LIN {X 0,Y 247.434,Z 446.734,A -85,B 0,C 180,E1 -19045.448,E2 -19045.448} C_VEL
LIN {X 0,Y 248.278,Z 445.373,A -85,B 0,C 180,E1 -19048.116,E2 -19048.116} C_VEL
LIN {X 0,Y 249.454,Z 442.811,A -85,B 0,C 180,E1 -19050.842,E2 -19050.842} C_VEL
LIN {X 0,Y 251.057,Z 438.873,A -85,B 0,C 180,E1 -19053.598,E2 -19053.598} C_VEL
LIN {X 0,Y 253.141,Z 433.443,A -85,B 0,C 180,E1 -19056.36,E2 -19056.36} C_VEL
LIN {X 0,Y 255.295,Z 427.674,A -85,B 0,C 180,E1 -19058.608,E2 -19058.608} C_VEL
LIN {X 0,Y 257.786,Z 420.296,A -85,B 0,C 180,E1 -19060.904,E2 -19060.904} C_VEL
LIN {X 0,Y 260.58,Z 411.115,A -85,B 0,C 180,E1 -19063.147,E2 -19063.147} C_VEL
LIN {X 0,Y 263.573,Z 400.733,A -85,B 0,C 180,E1 -19065.13,E2 -19065.13} C_VEL
LIN {X 0,Y 266.276,Z 389.982,A -85,B 0,C 180,E1 -19066.742,E2 -19066.742} C_VEL
LIN {X 0,Y 268.643,Z 378.487,A -85,B 0,C 180,E1 -19068.111,E2 -19068.111} C_VEL
LIN {X 0,Y 270.76,Z 365.913,A -85,B 0,C 180,E1 -19069.248,E2 -19069.248} C_VEL
LIN {X 0,Y 272.299,Z 353.044,A -85,B 0,C 180,E1 -19070.095,E2 -19070.095} C_VEL
LIN {X 0,Y 273.399,Z 340.201,A -85,B 0,C 180,E1 -19070.646,E2 -19070.646} C_VEL
LIN {X 0,Y 276.818,Z 284.839,A -85,B 0,C 180,E1 -19072.41,E2 -19072.41} C_VEL
LIN {X 0,Y 272.206,Z 274.812,A -85,B 0,C 180,E1 -19073.807,E2 -19073.807} C_VEL
LIN {X 0,Y 266.984,Z 265.08,A -85,B 0,C 180,E1 -19075.436,E2 -19075.436} C_VEL
LIN {X 0,Y 262.474,Z 257.861,A -85,B 0,C 180,E1 -19076.931,E2 -19076.931} C_VEL
LIN {X 0,Y 255.943,Z 247.889,A -85,B 0,C 180,E1 -19079.312,E2 -19079.312} C_VEL
LIN {X 0,Y 252.331,Z 243.094,A -85,B 0,C 180,E1 -19080.75,E2 -19080.75} C_VEL
LIN {X 0,Y 250.81,Z 241.467,A -85,B 0,C 180,E1 -19081.366,E2 -19081.366} C_VEL
LIN {X 0,Y 249.325,Z 240.348,A -85,B 0,C 180,E1 -19081.963,E2 -19081.963} C_VEL
LIN {X 0,Y 244.214,Z 240.449,A -85,B 0,C 180,E1 -19084.001,E2 -19084.001} C_VEL
LIN {X 0,Y 242.5,Z 239.911,A -85,B 0,C 180,E1 -19085.228,E2 -19085.228} C_VEL
LIN {X 0,Y 242.285,Z 239.3,A -85,B 0,C 180,E1 -19085.875,E2 -19085.875} C_VEL
LIN {X 0,Y 242.288,Z 239.303,A -85,B 0,C 180,E1 -19089.556,E2 -19089.556} C_VEL
LIN {X 0,Y 242.106,Z 239.323,A -85,B 0,C 180,E1 -19093.429,E2 -19093.429} C_VEL
LIN {X 0,Y 242.079,Z 239.323,A -85,B 0,C 180,E1 -19096.878,E2 -19096.878} C_VEL
LIN {X 0,Y 241.965,Z 239.346,A -85,B 0,C 180,E1 -19102.185,E2 -19102.185} C_VEL
LIN {X 0,Y 242.03,Z 239.332,A -85,B 0,C 180,E1 -19105.832,E2 -19105.832} C_VEL
LIN {X 0,Y 241.955,Z 239.338,A -85,B 0,C 180,E1 -19109.591,E2 -19109.591} C_VEL
LIN {X 0,Y 241.95,Z 239.343,A -85,B 0,C 180,E1 -19113.498,E2 -19113.498} C_VEL
LIN {X 0,Y 241.978,Z 239.412,A -85,B 0,C 180,E1 -19118.102,E2 -19118.102} C_VEL
LIN {X 0,Y 243.913,Z 244.836,A -85,B 0,C 180,E1 -19122.62,E2 -19122.62} C_VEL
LIN {X 0,Y 246.041,Z 251.254,A -85,B 0,C 180,E1 -19126.866,E2 -19126.866} C_VEL
LIN {X 0,Y 249.47,Z 256.649,A -85,B 0,C 180,E1 -19128.448,E2 -19128.448} C_VEL
LIN {X 0,Y 250.911,Z 258.872,A -85,B 0,C 180,E1 -19129.069,E2 -19129.069} C_VEL
LIN {X 0,Y 254.41,Z 264.527,A -85,B 0,C 180,E1 -19130.496,E2 -19130.496} C_VEL
LIN {X 0,Y 257.98,Z 270.888,A -85,B 0,C 180,E1 -19131.875,E2 -19131.875} C_VEL
LIN {X 0,Y 262.221,Z 279.028,A -85,B 0,C 180,E1 -19133.4,E2 -19133.4} C_VEL
LIN {X 0,Y 267,Z 289.735,A -85,B 0,C 180,E1 -19135.057,E2 -19135.057} C_VEL
LIN {X 0,Y 267.899,Z 292.556,A -85,B 0,C 180,E1 -19135.388,E2 -19135.388} C_VEL
LIN {X 0,Y 269.758,Z 308.366,A -85,B 0,C 180,E1 -19136.523,E2 -19136.523} C_VEL
LIN {X 0,Y 270.142,Z 313.745,A -85,B 0,C 180,E1 -19136.851,E2 -19136.851} C_VEL
LIN {X 0,Y 266.746,Z 363.722,A -85,B 0,C 180,E1 -19138.482,E2 -19138.482} C_VEL
LIN {X 0,Y 265.058,Z 377.664,A -85,B 0,C 180,E1 -19139.202,E2 -19139.202} C_VEL
LIN {X 0,Y 262.799,Z 390.364,A -85,B 0,C 180,E1 -19140.13,E2 -19140.13} C_VEL
LIN {X 0,Y 260.117,Z 402.51,A -85,B 0,C 180,E1 -19141.345,E2 -19141.345} C_VEL
LIN {X 0,Y 257.264,Z 413.548,A -85,B 0,C 180,E1 -19142.772,E2 -19142.772} C_VEL
LIN {X 0,Y 254.38,Z 423.635,A -85,B 0,C 180,E1 -19144.428,E2 -19144.428} C_VEL
LIN {X 0,Y 251.149,Z 433.64,A -85,B 0,C 180,E1 -19146.502,E2 -19146.502} C_VEL
LIN {X 0,Y 248.189,Z 442.707,A -85,B 0,C 180,E1 -19148.881,E2 -19148.881} C_VEL
LIN {X 0,Y 245.728,Z 449.849,A -85,B 0,C 180,E1 -19151.256,E2 -19151.256} C_VEL
LIN {X 0,Y 244.09,Z 454.725,A -85,B 0,C 180,E1 -19153.268,E2 -19153.268} C_VEL
LIN {X 0,Y 242.262,Z 459.556,A -85,B 0,C 180,E1 -19155.726,E2 -19155.726} C_VEL
LIN {X 0,Y 241.102,Z 463.286,A -85,B 0,C 180,E1 -19158.228,E2 -19158.228} C_VEL
LIN {X 0,Y 240.531,Z 465.241,A -85,B 0,C 180,E1 -19159.904,E2 -19159.904} C_VEL
LIN {X 0,Y 239.9,Z 467.837,A -85,B 0,C 180,E1 -19163.271,E2 -19163.271} C_VEL
LIN {X 0,Y 239.811,Z 468.612,A -85,B 0,C 180,E1 -19165.156,E2 -19165.156} C_VEL
LIN {X 0,Y 239.87,Z 468.846,A -85,B 0,C 180,E1 -19166.641,E2 -19166.641} C_VEL
LIN {X 0,Y 239.974,Z 468.704,A -85,B 0,C 180,E1 -19168.322,E2 -19168.322} C_VEL
LIN {X 0,Y 240.024,Z 468.154,A -85,B 0,C 180,E1 -19170,E2 -19170} C_VEL
LIN {X 0,Y 240.005,Z 467.189,A -85,B 0,C 180,E1 -19171.678,E2 -19171.678} C_VEL
LIN {X 0,Y 239.998,Z 465.777,A -85,B 0,C 180,E1 -19173.357,E2 -19173.357} C_VEL
LIN {X 0,Y 240.032,Z 463.373,A -85,B 0,C 180,E1 -19175.432,E2 -19175.432} C_VEL
LIN {X 0,Y 240.199,Z 458.645,A -85,B 0,C 180,E1 -19178.411,E2 -19178.411} C_VEL
LIN {X 0,Y 240.795,Z 452.239,A -85,B 0,C 180,E1 -19181.361,E2 -19181.361} C_VEL
LIN {X 0,Y 241.75,Z 445.225,A -85,B 0,C 180,E1 -19183.875,E2 -19183.875} C_VEL
LIN {X 0,Y 242.768,Z 438.024,A -85,B 0,C 180,E1 -19185.961,E2 -19185.961} C_VEL
LIN {X 0,Y 244.201,Z 428.768,A -85,B 0,C 180,E1 -19188.136,E2 -19188.136} C_VEL
LIN {X 0,Y 245.718,Z 418.531,A -85,B 0,C 180,E1 -19190.071,E2 -19190.071} C_VEL
LIN {X 0,Y 247.301,Z 407.905,A -85,B 0,C 180,E1 -19191.679,E2 -19191.679} C_VEL
LIN {X 0,Y 248.892,Z 396.173,A -85,B 0,C 180,E1 -19193.063,E2 -19193.063} C_VEL
LIN {X 0,Y 250.367,Z 382.933,A -85,B 0,C 180,E1 -19194.235,E2 -19194.235} C_VEL
LIN {X 0,Y 251.516,Z 369.594,A -85,B 0,C 180,E1 -19195.053,E2 -19195.053} C_VEL
LIN {X 0,Y 252.294,Z 352.667,A -85,B 0,C 180,E1 -19195.688,E2 -19195.688} C_VEL
LIN {X 0,Y 253.806,Z 307.843,A -85,B 0,C 180,E1 -19197.169,E2 -19197.169} C_VEL
LIN {X 0,Y 248.709,Z 266.187,A -85,B 0,C 180,E1 -19199.124,E2 -19199.124} C_VEL
LIN {X 0,Y 245.747,Z 257.13,A -85,B 0,C 180,E1 -19199.767,E2 -19199.767} C_VEL
LIN {X 0,Y 243.216,Z 244.807,A -85,B 0,C 180,E1 -19204.291,E2 -19204.291} C_VEL
LIN {X 0,Y 242.051,Z 239.335,A -85,B 0,C 180,E1 -19206.417,E2 -19206.417} C_VEL
LIN {X 0,Y 241.91,Z 239.35,A -85,B 0,C 180,E1 -19210.943,E2 -19210.943} C_VEL
LIN {X 0,Y 241.905,Z 239.355,A -85,B 0,C 180,E1 -19214.201,E2 -19214.201} C_VEL
LIN {X 0,Y 241.915,Z 239.352,A -85,B 0,C 180,E1 -19218.072,E2 -19218.072} C_VEL
LIN {X 0,Y 241.971,Z 239.342,A -85,B 0,C 180,E1 -19222.414,E2 -19222.414} C_VEL
LIN {X 0,Y 241.949,Z 239.343,A -85,B 0,C 180,E1 -19226.502,E2 -19226.502} C_VEL
LIN {X 0,Y 241.964,Z 239.343,A -85,B 0,C 180,E1 -19230.607,E2 -19230.607} C_VEL
LIN {X 0,Y 242.029,Z 239.331,A -85,B 0,C 180,E1 -19234.178,E2 -19234.178} C_VEL
LIN {X 0,Y 241.968,Z 239.343,A -85,B 0,C 180,E1 -19238.332,E2 -19238.332} C_VEL
LIN {X 0,Y 242.089,Z 239.32,A -85,B 0,C 180,E1 -19243.316,E2 -19243.316} C_VEL
LIN {X 0,Y 242.138,Z 239.32,A -85,B 0,C 180,E1 -19248.277,E2 -19248.277} C_VEL
LIN {X 0,Y 242.363,Z 239.294,A -85,B 0,C 180,E1 -19251.663,E2 -19251.663} C_VEL
LIN {X 0,Y 242.386,Z 239.29,A -85,B 0,C 180,E1 -19253.339,E2 -19253.339} C_VEL
LIN {X 0,Y 242.599,Z 239.251,A -85,B 0,C 180,E1 -19258.339,E2 -19258.339} C_VEL
LIN {X 0,Y 242.601,Z 239.255,A -85,B 0,C 180,E1 -19261.659,E2 -19261.659} C_VEL
LIN {X 0,Y 242.379,Z 239.292,A -85,B 0,C 180,E1 -19266.797,E2 -19266.797} C_VEL
LIN {X 0,Y 242.234,Z 239.309,A -85,B 0,C 180,E1 -19270.024,E2 -19270.024} C_VEL
LIN {X 0,Y 242.112,Z 239.314,A -85,B 0,C 180,E1 -19275.144,E2 -19275.144} C_VEL
LIN {X 0,Y 242.057,Z 239.312,A -85,B 0,C 180,E1 -19278.625,E2 -19278.625} C_VEL
LIN {X 0,Y 242.049,Z 239.322,A -85,B 0,C 180,E1 -19282.176,E2 -19282.176} C_VEL
LIN {X 0,Y 242.044,Z 239.33,A -85,B 0,C 180,E1 -19285.84,E2 -19285.84} C_VEL
LIN {X 0,Y 242.007,Z 239.337,A -85,B 0,C 180,E1 -19289.583,E2 -19289.583} C_VEL
LIN {X 0,Y 241.96,Z 239.34,A -85,B 0,C 180,E1 -19293.495,E2 -19293.495} C_VEL
LIN {X 0,Y 241.98,Z 239.329,A -85,B 0,C 180,E1 -19297.583,E2 -19297.583} C_VEL
LIN {X 0,Y 241.964,Z 239.331,A -85,B 0,C 180,E1 -19301.916,E2 -19301.916} C_VEL
LIN {X 0,Y 241.921,Z 239.347,A -85,B 0,C 180,E1 -19305.802,E2 -19305.802} C_VEL
LIN {X 0,Y 241.943,Z 239.347,A -85,B 0,C 180,E1 -19310.284,E2 -19310.284} C_VEL
LIN {X 0,Y 241.976,Z 239.335,A -85,B 0,C 180,E1 -19314.492,E2 -19314.492} C_VEL
LIN {X 0,Y 241.965,Z 239.333,A -85,B 0,C 180,E1 -19318.483,E2 -19318.483} C_VEL
LIN {X 0,Y 242.003,Z 239.338,A -85,B 0,C 180,E1 -19322.316,E2 -19322.316} C_VEL
LIN {X 0,Y 242.051,Z 239.334,A -85,B 0,C 180,E1 -19326.018,E2 -19326.018} C_VEL
LIN {X 0,Y 242.032,Z 239.331,A -85,B 0,C 180,E1 -19329.61,E2 -19329.61} C_VEL
LIN {X 0,Y 242.159,Z 239.316,A -85,B 0,C 180,E1 -19333.28,E2 -19333.28} C_VEL
LIN {X 0,Y 242.184,Z 239.314,A -85,B 0,C 180,E1 -19338.281,E2 -19338.281} C_VEL
LIN {X 0,Y 242.424,Z 239.287,A -85,B 0,C 180,E1 -19341.667,E2 -19341.667} C_VEL
LIN {X 0,Y 242.257,Z 239.31,A -85,B 0,C 180,E1 -19345.008,E2 -19345.008} C_VEL
LIN {X 0,Y 242.635,Z 239.258,A -85,B 0,C 180,E1 -19348.341,E2 -19348.341} C_VEL
LIN {X 0,Y 242.635,Z 239.259,A -85,B 0,C 180,E1 -19351.66,E2 -19351.66} C_VEL
LIN {X 0,Y 242.423,Z 239.287,A -85,B 0,C 180,E1 -19356.659,E2 -19356.659} C_VEL
LIN {X 0,Y 242.265,Z 239.307,A -85,B 0,C 180,E1 -19360.023,E2 -19360.023} C_VEL
LIN {X 0,Y 242.163,Z 239.322,A -85,B 0,C 180,E1 -19365.139,E2 -19365.139} C_VEL
LIN {X 0,Y 242.067,Z 239.332,A -85,B 0,C 180,E1 -19369.503,E2 -19369.503} C_VEL
LIN {X 0,Y 242.098,Z 239.466,A -85,B 0,C 180,E1 -19370.163,E2 -19370.163} C_VEL
LIN {X 0,Y 247.724,Z 253.276,A -85,B 0,C 180,E1 -19371.215,E2 -19371.215} C_VEL
LIN {X 0,Y 253.573,Z 269.164,A -85,B 0,C 180,E1 -19372.309,E2 -19372.309} C_VEL
LIN {X 0,Y 254.862,Z 273.057,A -85,B 0,C 180,E1 -19372.559,E2 -19372.559} C_VEL
LIN {X 0,Y 252.021,Z 343.618,A -85,B 0,C 180,E1 -19374.889,E2 -19374.889} C_VEL
LIN {X 0,Y 251.08,Z 357.249,A -85,B 0,C 180,E1 -19375.654,E2 -19375.654} C_VEL
LIN {X 0,Y 250.037,Z 370.169,A -85,B 0,C 180,E1 -19376.723,E2 -19376.723} C_VEL
LIN {X 0,Y 248.619,Z 382.874,A -85,B 0,C 180,E1 -19378.143,E2 -19378.143} C_VEL
LIN {X 0,Y 247.293,Z 393.032,A -85,B 0,C 180,E1 -19379.587,E2 -19379.587} C_VEL
LIN {X 0,Y 245.776,Z 403.642,A -85,B 0,C 180,E1 -19381.462,E2 -19381.462} C_VEL
LIN {X 0,Y 244.339,Z 412.802,A -85,B 0,C 180,E1 -19383.475,E2 -19383.475} C_VEL
LIN {X 0,Y 242.893,Z 421.687,A -85,B 0,C 180,E1 -19385.889,E2 -19385.889} C_VEL
LIN {X 0,Y 241.795,Z 428.792,A -85,B 0,C 180,E1 -19388.301,E2 -19388.301} C_VEL
LIN {X 0,Y 240.966,Z 434.411,A -85,B 0,C 180,E1 -19390.685,E2 -19390.685} C_VEL
LIN {X 0,Y 240.445,Z 438.85,A -85,B 0,C 180,E1 -19393.053,E2 -19393.053} C_VEL
LIN {X 0,Y 239.996,Z 442.182,A -85,B 0,C 180,E1 -19395.348,E2 -19395.348} C_VEL
LIN {X 0,Y 239.735,Z 444.602,A -85,B 0,C 180,E1 -19397.604,E2 -19397.604} C_VEL
LIN {X 0,Y 239.645,Z 446.243,A -85,B 0,C 180,E1 -19399.821,E2 -19399.821} C_VEL
LIN {X 0,Y 239.806,Z 447.23,A -85,B 0,C 180,E1 -19402.298,E2 -19402.298} C_VEL
LIN {X 0,Y 240.228,Z 447.289,A -85,B 0,C 180,E1 -19404.991,E2 -19404.991} C_VEL
LIN {X 0,Y 241.028,Z 446.267,A -85,B 0,C 180,E1 -19407.726,E2 -19407.726} C_VEL
LIN {X 0,Y 242.178,Z 444.088,A -85,B 0,C 180,E1 -19410.517,E2 -19410.517} C_VEL
LIN {X 0,Y 243.783,Z 440.637,A -85,B 0,C 180,E1 -19413.329,E2 -19413.329} C_VEL
LIN {X 0,Y 246.062,Z 435.194,A -85,B 0,C 180,E1 -19416.431,E2 -19416.431} C_VEL
LIN {X 0,Y 248.473,Z 429.163,A -85,B 0,C 180,E1 -19418.955,E2 -19418.955} C_VEL
LIN {X 0,Y 251.308,Z 421.317,A -85,B 0,C 180,E1 -19421.515,E2 -19421.515} C_VEL
LIN {X 0,Y 254.172,Z 412.662,A -85,B 0,C 180,E1 -19423.743,E2 -19423.743} C_VEL
LIN {X 0,Y 257.286,Z 402.561,A -85,B 0,C 180,E1 -19425.769,E2 -19425.769} C_VEL
LIN {X 0,Y 259.926,Z 392.988,A -85,B 0,C 180,E1 -19427.295,E2 -19427.295} C_VEL
LIN {X 0,Y 262.588,Z 381.11,A -85,B 0,C 180,E1 -19428.812,E2 -19428.812} C_VEL
LIN {X 0,Y 264.792,Z 369.498,A -85,B 0,C 180,E1 -19429.931,E2 -19429.931} C_VEL
LIN {X 0,Y 266.554,Z 356.371,A -85,B 0,C 180,E1 -19430.898,E2 -19430.898} C_VEL
LIN {X 0,Y 267.891,Z 342.608,A -85,B 0,C 180,E1 -19431.545,E2 -19431.545} C_VEL
LIN {X 0,Y 271.618,Z 287.449,A -85,B 0,C 180,E1 -19433.342,E2 -19433.342} C_VEL
LIN {X 0,Y 266.636,Z 276.755,A -85,B 0,C 180,E1 -19434.933,E2 -19434.933} C_VEL
LIN {X 0,Y 261.493,Z 267.258,A -85,B 0,C 180,E1 -19436.682,E2 -19436.682} C_VEL
LIN {X 0,Y 253.706,Z 254.952,A -85,B 0,C 180,E1 -19439.567,E2 -19439.567} C_VEL
LIN {X 0,Y 249.474,Z 249.158,A -85,B 0,C 180,E1 -19441.312,E2 -19441.312} C_VEL
LIN {X 0,Y 247.381,Z 246.516,A -85,B 0,C 180,E1 -19442.24,E2 -19442.24} C_VEL
LIN {X 0,Y 245.331,Z 244.219,A -85,B 0,C 180,E1 -19443.182,E2 -19443.182} C_VEL
LIN {X 0,Y 243.211,Z 242.091,A -85,B 0,C 180,E1 -19444.195,E2 -19444.195} C_VEL
LIN {X 0,Y 242.531,Z 240.662,A -85,B 0,C 180,E1 -19444.675,E2 -19444.675} C_VEL
LIN {X 0,Y 242.285,Z 239.3,A -85,B 0,C 180,E1 -19445.875,E2 -19445.875} C_VEL
LIN {X 0,Y 241.688,Z 239.381,A -85,B 0,C 180,E1 -19447.263,E2 -19447.263} C_VEL
LIN {X 0,Y 240.082,Z 239.578,A -85,B 0,C 180,E1 -19448.623,E2 -19448.623} C_VEL
LIN {X 0,Y 236.204,Z 240.055,A -85,B 0,C 180,E1 -19451.362,E2 -19451.362} C_VEL
LIN {X 0,Y 235.113,Z 240.199,A -85,B 0,C 180,E1 -19452.795,E2 -19452.795} C_VEL
LIN {X 0,Y 235.03,Z 240.199,A -85,B 0,C 180,E1 -19453.282,E2 -19453.282} C_VEL
LIN {X 0,Y 234.987,Z 240.206,A -85,B 0,C 180,E1 -19457.403,E2 -19457.403} C_VEL
LIN {X 0,Y 234.931,Z 240.223,A -85,B 0,C 180,E1 -19461.987,E2 -19461.987} C_VEL
LIN {X 0,Y 234.962,Z 240.21,A -85,B 0,C 180,E1 -19466.202,E2 -19466.202} C_VEL
LIN {X 0,Y 234.874,Z 240.223,A -85,B 0,C 180,E1 -19470.577,E2 -19470.577} C_VEL
LIN {X 0,Y 234.902,Z 240.364,A -85,B 0,C 180,E1 -19474.43,E2 -19474.43} C_VEL
LIN {X 0,Y 236.327,Z 244.216,A -85,B 0,C 180,E1 -19478.647,E2 -19478.647} C_VEL
LIN {X 0,Y 238.304,Z 249.77,A -85,B 0,C 180,E1 -19483.29,E2 -19483.29} C_VEL
LIN {X 0,Y 238.701,Z 250.699,A -85,B 0,C 180,E1 -19483.782,E2 -19483.782} C_VEL
LIN {X 0,Y 242.195,Z 255.987,A -85,B 0,C 180,E1 -19485.722,E2 -19485.722} C_VEL
LIN {X 0,Y 243.536,Z 257.884,A -85,B 0,C 180,E1 -19486.391,E2 -19486.391} C_VEL
LIN {X 0,Y 247.667,Z 264.331,A -85,B 0,C 180,E1 -19488.345,E2 -19488.345} C_VEL
LIN {X 0,Y 250.972,Z 269.919,A -85,B 0,C 180,E1 -19489.778,E2 -19489.778} C_VEL
LIN {X 0,Y 254.538,Z 276.479,A -85,B 0,C 180,E1 -19491.234,E2 -19491.234} C_VEL
LIN {X 0,Y 258.642,Z 284.708,A -85,B 0,C 180,E1 -19492.796,E2 -19492.796} C_VEL
LIN {X 0,Y 262.568,Z 293.805,A -85,B 0,C 180,E1 -19494.25,E2 -19494.25} C_VEL
LIN {X 0,Y 263.191,Z 296.443,A -85,B 0,C 180,E1 -19494.53,E2 -19494.53} C_VEL
LIN {X 0,Y 264.967,Z 313.222,A -85,B 0,C 180,E1 -19495.738,E2 -19495.738} C_VEL
LIN {X 0,Y 264.011,Z 329.304,A -85,B 0,C 180,E1 -19496.306,E2 -19496.306} C_VEL
LIN {X 0,Y 261.401,Z 364.197,A -85,B 0,C 180,E1 -19497.475,E2 -19497.475} C_VEL
LIN {X 0,Y 259.74,Z 377.087,A -85,B 0,C 180,E1 -19498.159,E2 -19498.159} C_VEL
LIN {X 0,Y 257.59,Z 388.754,A -85,B 0,C 180,E1 -19499.008,E2 -19499.008} C_VEL
LIN {X 0,Y 254.793,Z 401.155,A -85,B 0,C 180,E1 -19500.235,E2 -19500.235} C_VEL
LIN {X 0,Y 251.42,Z 413.648,A -85,B 0,C 180,E1 -19501.858,E2 -19501.858} C_VEL
LIN {X 0,Y 248.401,Z 423.636,A -85,B 0,C 180,E1 -19503.54,E2 -19503.54} C_VEL
LIN {X 0,Y 245.331,Z 432.76,A -85,B 0,C 180,E1 -19505.459,E2 -19505.459} C_VEL
LIN {X 0,Y 242.106,Z 441.733,A -85,B 0,C 180,E1 -19507.831,E2 -19507.831} C_VEL
LIN {X 0,Y 239.435,Z 449.019,A -85,B 0,C 180,E1 -19510.274,E2 -19510.274} C_VEL
LIN {X 0,Y 237.291,Z 454.933,A -85,B 0,C 180,E1 -19512.774,E2 -19512.774} C_VEL
LIN {X 0,Y 235.374,Z 459.645,A -85,B 0,C 180,E1 -19515.299,E2 -19515.299} C_VEL
LIN {X 0,Y 234.118,Z 463.277,A -85,B 0,C 180,E1 -19517.871,E2 -19517.871} C_VEL
LIN {X 0,Y 233.101,Z 466.566,A -85,B 0,C 180,E1 -19521.33,E2 -19521.33} C_VEL
LIN {X 0,Y 232.744,Z 468.27,A -85,B 0,C 180,E1 -19524.803,E2 -19524.803} C_VEL
LIN {X 0,Y 232.769,Z 468.485,A -85,B 0,C 180,E1 -19526.538,E2 -19526.538} C_VEL
LIN {X 0,Y 232.9,Z 468.298,A -85,B 0,C 180,E1 -19528.271,E2 -19528.271} C_VEL
LIN {X 0,Y 232.951,Z 467.702,A -85,B 0,C 180,E1 -19530,E2 -19530} C_VEL
LIN {X 0,Y 232.935,Z 466.683,A -85,B 0,C 180,E1 -19531.729,E2 -19531.729} C_VEL
LIN {X 0,Y 232.916,Z 465.178,A -85,B 0,C 180,E1 -19533.459,E2 -19533.459} C_VEL
LIN {X 0,Y 232.949,Z 462.198,A -85,B 0,C 180,E1 -19535.974,E2 -19535.974} C_VEL
LIN {X 0,Y 233.16,Z 457.827,A -85,B 0,C 180,E1 -19538.667,E2 -19538.667} C_VEL
LIN {X 0,Y 233.781,Z 451.296,A -85,B 0,C 180,E1 -19541.706,E2 -19541.706} C_VEL
LIN {X 0,Y 234.838,Z 444.123,A -85,B 0,C 180,E1 -19544.292,E2 -19544.292} C_VEL
LIN {X 0,Y 235.922,Z 436.754,A -85,B 0,C 180,E1 -19546.437,E2 -19546.437} C_VEL
LIN {X 0,Y 237.086,Z 429.047,A -85,B 0,C 180,E1 -19548.3,E2 -19548.3} C_VEL
LIN {X 0,Y 238.639,Z 419.2,A -85,B 0,C 180,E1 -19550.243,E2 -19550.243} C_VEL
LIN {X 0,Y 240.253,Z 408.792,A -85,B 0,C 180,E1 -19551.896,E2 -19551.896} C_VEL
LIN {X 0,Y 241.832,Z 397.47,A -85,B 0,C 180,E1 -19553.323,E2 -19553.323} C_VEL
LIN {X 0,Y 243.174,Z 386.002,A -85,B 0,C 180,E1 -19554.431,E2 -19554.431} C_VEL
LIN {X 0,Y 244.474,Z 372.468,A -85,B 0,C 180,E1 -19555.37,E2 -19555.37} C_VEL
LIN {X 0,Y 245.315,Z 359.267,A -85,B 0,C 180,E1 -19555.96,E2 -19555.96} C_VEL
LIN {X 0,Y 247.135,Z 308.763,A -85,B 0,C 180,E1 -19557.679,E2 -19557.679} C_VEL
LIN {X 0,Y 242.157,Z 267.874,A -85,B 0,C 180,E1 -19559.649,E2 -19559.649} C_VEL
LIN {X 0,Y 238.436,Z 256.827,A -85,B 0,C 180,E1 -19560.467,E2 -19560.467} C_VEL
LIN {X 0,Y 236.014,Z 244.954,A -85,B 0,C 180,E1 -19564.971,E2 -19564.971} C_VEL
LIN {X 0,Y 234.987,Z 240.215,A -85,B 0,C 180,E1 -19566.867,E2 -19566.867} C_VEL
LIN {X 0,Y 234.862,Z 240.231,A -85,B 0,C 180,E1 -19571.573,E2 -19571.573} C_VEL
LIN {X 0,Y 234.87,Z 240.232,A -85,B 0,C 180,E1 -19575.895,E2 -19575.895} C_VEL
LIN {X 0,Y 234.856,Z 240.229,A -85,B 0,C 180,E1 -19578.826,E2 -19578.826} C_VEL
LIN {X 0,Y 234.91,Z 240.223,A -85,B 0,C 180,E1 -19583.247,E2 -19583.247} C_VEL
LIN {X 0,Y 234.912,Z 240.222,A -85,B 0,C 180,E1 -19587.417,E2 -19587.417} C_VEL
LIN {X 0,Y 234.894,Z 240.226,A -85,B 0,C 180,E1 -19591.398,E2 -19591.398} C_VEL
LIN {X 0,Y 234.945,Z 240.215,A -85,B 0,C 180,E1 -19595.241,E2 -19595.241} C_VEL
LIN {X 0,Y 234.918,Z 240.223,A -85,B 0,C 180,E1 -19598.96,E2 -19598.96} C_VEL
LIN {X 0,Y 235.03,Z 240.201,A -85,B 0,C 180,E1 -19603.092,E2 -19603.092} C_VEL
LIN {X 0,Y 235.07,Z 240.2,A -85,B 0,C 180,E1 -19607.919,E2 -19607.919} C_VEL
LIN {X 0,Y 235.292,Z 240.176,A -85,B 0,C 180,E1 -19611.41,E2 -19611.41} C_VEL
LIN {X 0,Y 235.336,Z 240.169,A -85,B 0,C 180,E1 -19613.139,E2 -19613.139} C_VEL
LIN {X 0,Y 235.559,Z 240.127,A -85,B 0,C 180,E1 -19618.29,E2 -19618.29} C_VEL
LIN {X 0,Y 235.561,Z 240.131,A -85,B 0,C 180,E1 -19621.709,E2 -19621.709} C_VEL
LIN {X 0,Y 235.339,Z 240.171,A -85,B 0,C 180,E1 -19626.86,E2 -19626.86} C_VEL
LIN {X 0,Y 235.183,Z 240.188,A -85,B 0,C 180,E1 -19630.328,E2 -19630.328} C_VEL
LIN {X 0,Y 235.067,Z 240.189,A -85,B 0,C 180,E1 -19635.609,E2 -19635.609} C_VEL
LIN {X 0,Y 235.003,Z 240.189,A -85,B 0,C 180,E1 -19639.205,E2 -19639.205} C_VEL
LIN {X 0,Y 234.978,Z 240.207,A -85,B 0,C 180,E1 -19642.88,E2 -19642.88} C_VEL
LIN {X 0,Y 234.947,Z 240.218,A -85,B 0,C 180,E1 -19646.659,E2 -19646.659} C_VEL
LIN {X 0,Y 234.909,Z 240.223,A -85,B 0,C 180,E1 -19650.57,E2 -19650.57} C_VEL
LIN {X 0,Y 234.913,Z 240.215,A -85,B 0,C 180,E1 -19654.64,E2 -19654.64} C_VEL
LIN {X 0,Y 234.949,Z 240.196,A -85,B 0,C 180,E1 -19658.955,E2 -19658.955} C_VEL
LIN {X 0,Y 234.943,Z 240.209,A -85,B 0,C 180,E1 -19663.472,E2 -19663.472} C_VEL
LIN {X 0,Y 234.87,Z 240.228,A -85,B 0,C 180,E1 -19668.423,E2 -19668.423} C_VEL
LIN {X 0,Y 234.905,Z 240.222,A -85,B 0,C 180,E1 -19671.081,E2 -19671.081} C_VEL
LIN {X 0,Y 234.919,Z 240.214,A -85,B 0,C 180,E1 -19675.365,E2 -19675.365} C_VEL
LIN {X 0,Y 234.923,Z 240.211,A -85,B 0,C 180,E1 -19679.435,E2 -19679.435} C_VEL
LIN {X 0,Y 234.987,Z 240.216,A -85,B 0,C 180,E1 -19683.796,E2 -19683.796} C_VEL
LIN {X 0,Y 235.006,Z 240.207,A -85,B 0,C 180,E1 -19688.972,E2 -19688.972} C_VEL
LIN {X 0,Y 235.092,Z 240.195,A -85,B 0,C 180,E1 -19693.061,E2 -19693.061} C_VEL
LIN {X 0,Y 235.144,Z 240.192,A -85,B 0,C 180,E1 -19697.925,E2 -19697.925} C_VEL
LIN {X 0,Y 235.374,Z 240.163,A -85,B 0,C 180,E1 -19701.415,E2 -19701.415} C_VEL
LIN {X 0,Y 235.401,Z 240.163,A -85,B 0,C 180,E1 -19703.142,E2 -19703.142} C_VEL
LIN {X 0,Y 235.595,Z 240.135,A -85,B 0,C 180,E1 -19708.291,E2 -19708.291} C_VEL
LIN {X 0,Y 235.594,Z 240.136,A -85,B 0,C 180,E1 -19711.709,E2 -19711.709} C_VEL
LIN {X 0,Y 235.392,Z 240.163,A -85,B 0,C 180,E1 -19716.858,E2 -19716.858} C_VEL
LIN {X 0,Y 235.212,Z 240.186,A -85,B 0,C 180,E1 -19720.327,E2 -19720.327} C_VEL
LIN {X 0,Y 235.109,Z 240.199,A -85,B 0,C 180,E1 -19725.605,E2 -19725.605} C_VEL
LIN {X 0,Y 235.046,Z 240.207,A -85,B 0,C 180,E1 -19729.45,E2 -19729.45} C_VEL
LIN {X 0,Y 236.05,Z 243.081,A -85,B 0,C 180,E1 -19729.706,E2 -19729.706} C_VEL
LIN {X 0,Y 243.947,Z 262.287,A -85,B 0,C 180,E1 -19731.216,E2 -19731.216} C_VEL
LIN {X 0,Y 248.189,Z 274.662,A -85,B 0,C 180,E1 -19732.052,E2 -19732.052} C_VEL
LIN {X 0,Y 245.23,Z 344.259,A -85,B 0,C 180,E1 -19734.425,E2 -19734.425} C_VEL
LIN {X 0,Y 244.278,Z 357.597,A -85,B 0,C 180,E1 -19735.2,E2 -19735.2} C_VEL
LIN {X 0,Y 243.267,Z 369.85,A -85,B 0,C 180,E1 -19736.231,E2 -19736.231} C_VEL
LIN {X 0,Y 241.955,Z 381.443,A -85,B 0,C 180,E1 -19737.526,E2 -19737.526} C_VEL
LIN {X 0,Y 240.336,Z 393.701,A -85,B 0,C 180,E1 -19739.291,E2 -19739.291} C_VEL
LIN {X 0,Y 238.973,Z 403.015,A -85,B 0,C 180,E1 -19740.971,E2 -19740.971} C_VEL
LIN {X 0,Y 237.328,Z 413.061,A -85,B 0,C 180,E1 -19743.215,E2 -19743.215} C_VEL
LIN {X 0,Y 236.069,Z 420.758,A -85,B 0,C 180,E1 -19745.333,E2 -19745.333} C_VEL
LIN {X 0,Y 234.915,Z 427.886,A -85,B 0,C 180,E1 -19747.733,E2 -19747.733} C_VEL
LIN {X 0,Y 233.85,Z 434.849,A -85,B 0,C 180,E1 -19750.705,E2 -19750.705} C_VEL
LIN {X 0,Y 233.211,Z 440.074,A -85,B 0,C 180,E1 -19753.677,E2 -19753.677} C_VEL
LIN {X 0,Y 232.733,Z 443.641,A -85,B 0,C 180,E1 -19756.441,E2 -19756.441} C_VEL
LIN {X 0,Y 232.559,Z 445.958,A -85,B 0,C 180,E1 -19759.063,E2 -19759.063} C_VEL
LIN {X 0,Y 232.665,Z 447.329,A -85,B 0,C 180,E1 -19761.747,E2 -19761.747} C_VEL
LIN {X 0,Y 233.171,Z 447.696,A -85,B 0,C 180,E1 -19765.064,E2 -19765.064} C_VEL
LIN {X 0,Y 233.779,Z 447.06,A -85,B 0,C 180,E1 -19767.316,E2 -19767.316} C_VEL
LIN {X 0,Y 234.913,Z 445.277,A -85,B 0,C 180,E1 -19770.171,E2 -19770.171} C_VEL
LIN {X 0,Y 236.807,Z 441.593,A -85,B 0,C 180,E1 -19773.566,E2 -19773.566} C_VEL
LIN {X 0,Y 238.536,Z 437.849,A -85,B 0,C 180,E1 -19775.959,E2 -19775.959} C_VEL
LIN {X 0,Y 241.138,Z 431.842,A -85,B 0,C 180,E1 -19778.835,E2 -19778.835} C_VEL
LIN {X 0,Y 244.158,Z 424.436,A -85,B 0,C 180,E1 -19781.541,E2 -19781.541} C_VEL
LIN {X 0,Y 247.334,Z 415.513,A -85,B 0,C 180,E1 -19784.054,E2 -19784.054} C_VEL
LIN {X 0,Y 250.681,Z 405.604,A -85,B 0,C 180,E1 -19786.214,E2 -19786.214} C_VEL
LIN {X 0,Y 253.801,Z 394.988,A -85,B 0,C 180,E1 -19788.014,E2 -19788.014} C_VEL
LIN {X 0,Y 256.718,Z 383.058,A -85,B 0,C 180,E1 -19789.621,E2 -19789.621} C_VEL
LIN {X 0,Y 259.181,Z 371.085,A -85,B 0,C 180,E1 -19790.834,E2 -19790.834} C_VEL
LIN {X 0,Y 261.131,Z 357.847,A -85,B 0,C 180,E1 -19791.853,E2 -19791.853} C_VEL
LIN {X 0,Y 262.491,Z 345.193,A -85,B 0,C 180,E1 -19792.506,E2 -19792.506} C_VEL
LIN {X 0,Y 266.384,Z 289.809,A -85,B 0,C 180,E1 -19794.355,E2 -19794.355} C_VEL
LIN {X 0,Y 261.126,Z 278.567,A -85,B 0,C 180,E1 -19796.176,E2 -19796.176} C_VEL
LIN {X 0,Y 256.131,Z 269.685,A -85,B 0,C 180,E1 -19797.979,E2 -19797.979} C_VEL
LIN {X 0,Y 249.482,Z 259.174,A -85,B 0,C 180,E1 -19800.651,E2 -19800.651} C_VEL
LIN {X 0,Y 246.534,Z 255.089,A -85,B 0,C 180,E1 -19801.954,E2 -19801.954} C_VEL
LIN {X 0,Y 243.219,Z 250.835,A -85,B 0,C 180,E1 -19803.521,E2 -19803.521} C_VEL
LIN {X 0,Y 240.848,Z 248.444,A -85,B 0,C 180,E1 -19804.708,E2 -19804.708} C_VEL
LIN {X 0,Y 239.223,Z 246.142,A -85,B 0,C 180,E1 -19805.627,E2 -19805.627} C_VEL
LIN {X 0,Y 236.105,Z 242.651,A -85,B 0,C 180,E1 -19807.483,E2 -19807.483} C_VEL
LIN {X 0,Y 235.632,Z 241.553,A -85,B 0,C 180,E1 -19807.93,E2 -19807.93} C_VEL
LIN {X 0,Y 235.233,Z 240.182,A -85,B 0,C 180,E1 -19809.659,E2 -19809.659} C_VEL
LIN {X 0,Y 235.03,Z 240.199,A -85,B 0,C 180,E1 -19813.282,E2 -19813.282} C_VEL
LIN {X 0,Y 234.359,Z 240.287,A -85,B 0,C 180,E1 -19814.712,E2 -19814.712} C_VEL
LIN {X 0,Y 231.443,Z 240.647,A -85,B 0,C 180,E1 -19817.042,E2 -19817.042} C_VEL
LIN {X 0,Y 228.97,Z 240.965,A -85,B 0,C 180,E1 -19818.942,E2 -19818.942} C_VEL
LIN {X 0,Y 227.929,Z 241.086,A -85,B 0,C 180,E1 -19820.42,E2 -19820.42} C_VEL
LIN {X 0,Y 227.855,Z 241.095,A -85,B 0,C 180,E1 -19820.921,E2 -19820.921} C_VEL
LIN {X 0,Y 227.894,Z 241.094,A -85,B 0,C 180,E1 -19825.579,E2 -19825.579} C_VEL
LIN {X 0,Y 227.886,Z 241.306,A -85,B 0,C 180,E1 -19828.557,E2 -19828.557} C_VEL
LIN {X 0,Y 229.136,Z 244.378,A -85,B 0,C 180,E1 -19834.101,E2 -19834.101} C_VEL
LIN {X 0,Y 230.715,Z 249.085,A -85,B 0,C 180,E1 -19839.275,E2 -19839.275} C_VEL
LIN {X 0,Y 236.327,Z 257.048,A -85,B 0,C 180,E1 -19843.215,E2 -19843.215} C_VEL
LIN {X 0,Y 239.825,Z 262.361,A -85,B 0,C 180,E1 -19845.235,E2 -19845.235} C_VEL
LIN {X 0,Y 244.758,Z 270.283,A -85,B 0,C 180,E1 -19847.726,E2 -19847.726} C_VEL
LIN {X 0,Y 248.05,Z 276.159,A -85,B 0,C 180,E1 -19849.245,E2 -19849.245} C_VEL
LIN {X 0,Y 252.2,Z 284.054,A -85,B 0,C 180,E1 -19850.999,E2 -19850.999} C_VEL
LIN {X 0,Y 256.559,Z 293.721,A -85,B 0,C 180,E1 -19852.743,E2 -19852.743} C_VEL
LIN {X 0,Y 258.437,Z 298.792,A -85,B 0,C 180,E1 -19853.494,E2 -19853.494} C_VEL
LIN {X 0,Y 259.948,Z 314.794,A -85,B 0,C 180,E1 -19854.702,E2 -19854.702} C_VEL
LIN {X 0,Y 256.323,Z 363.55,A -85,B 0,C 180,E1 -19856.371,E2 -19856.371} C_VEL
LIN {X 0,Y 254.534,Z 376.807,A -85,B 0,C 180,E1 -19857.075,E2 -19857.075} C_VEL
LIN {X 0,Y 252.074,Z 389.464,A -85,B 0,C 180,E1 -19858.016,E2 -19858.016} C_VEL
LIN {X 0,Y 249.155,Z 401.568,A -85,B 0,C 180,E1 -19859.256,E2 -19859.256} C_VEL
LIN {X 0,Y 246.032,Z 412.58,A -85,B 0,C 180,E1 -19860.717,E2 -19860.717} C_VEL
LIN {X 0,Y 242.839,Z 422.661,A -85,B 0,C 180,E1 -19862.419,E2 -19862.419} C_VEL
LIN {X 0,Y 239.573,Z 431.887,A -85,B 0,C 180,E1 -19864.364,E2 -19864.364} C_VEL
LIN {X 0,Y 236.632,Z 439.583,A -85,B 0,C 180,E1 -19866.365,E2 -19866.365} C_VEL
LIN {X 0,Y 233.658,Z 447.18,A -85,B 0,C 180,E1 -19868.844,E2 -19868.844} C_VEL
LIN {X 0,Y 231.262,Z 453.345,A -85,B 0,C 180,E1 -19871.394,E2 -19871.394} C_VEL
LIN {X 0,Y 229.108,Z 458.291,A -85,B 0,C 180,E1 -19873.975,E2 -19873.975} C_VEL
LIN {X 0,Y 227.5,Z 462.154,A -85,B 0,C 180,E1 -19876.605,E2 -19876.605} C_VEL
LIN {X 0,Y 226.516,Z 465.017,A -85,B 0,C 180,E1 -19879.272,E2 -19879.272} C_VEL
LIN {X 0,Y 225.768,Z 467.403,A -85,B 0,C 180,E1 -19882.848,E2 -19882.848} C_VEL
LIN {X 0,Y 225.631,Z 468.076,A -85,B 0,C 180,E1 -19885.382,E2 -19885.382} C_VEL
LIN {X 0,Y 225.827,Z 467.891,A -85,B 0,C 180,E1 -19888.217,E2 -19888.217} C_VEL
LIN {X 0,Y 225.881,Z 467.251,A -85,B 0,C 180,E1 -19890,E2 -19890} C_VEL
LIN {X 0,Y 225.866,Z 466.143,A -85,B 0,C 180,E1 -19891.783,E2 -19891.783} C_VEL
LIN {X 0,Y 225.823,Z 463.64,A -85,B 0,C 180,E1 -19894.468,E2 -19894.468} C_VEL
LIN {X 0,Y 225.919,Z 460.063,A -85,B 0,C 180,E1 -19897.147,E2 -19897.147} C_VEL
LIN {X 0,Y 226.261,Z 455.292,A -85,B 0,C 180,E1 -19899.835,E2 -19899.835} C_VEL
LIN {X 0,Y 226.887,Z 449.187,A -85,B 0,C 180,E1 -19902.521,E2 -19902.521} C_VEL
LIN {X 0,Y 228.094,Z 441.572,A -85,B 0,C 180,E1 -19905.181,E2 -19905.181} C_VEL
LIN {X 0,Y 229.347,Z 433.767,A -85,B 0,C 180,E1 -19907.382,E2 -19907.382} C_VEL
LIN {X 0,Y 230.664,Z 425.565,A -85,B 0,C 180,E1 -19909.286,E2 -19909.286} C_VEL
LIN {X 0,Y 232.34,Z 414.963,A -85,B 0,C 180,E1 -19911.281,E2 -19911.281} C_VEL
LIN {X 0,Y 234.039,Z 403.568,A -85,B 0,C 180,E1 -19912.975,E2 -19912.975} C_VEL
LIN {X 0,Y 235.744,Z 391.921,A -85,B 0,C 180,E1 -19914.314,E2 -19914.314} C_VEL
LIN {X 0,Y 237.08,Z 379.309,A -85,B 0,C 180,E1 -19915.395,E2 -19915.395} C_VEL
LIN {X 0,Y 238.214,Z 365.561,A -85,B 0,C 180,E1 -19916.204,E2 -19916.204} C_VEL
LIN {X 0,Y 240.405,Z 309.426,A -85,B 0,C 180,E1 -19918.204,E2 -19918.204} C_VEL
LIN {X 0,Y 235.733,Z 270.066,A -85,B 0,C 180,E1 -19920.163,E2 -19920.163} C_VEL
LIN {X 0,Y 231.136,Z 256.525,A -85,B 0,C 180,E1 -19921.19,E2 -19921.19} C_VEL
LIN {X 0,Y 229.009,Z 246.127,A -85,B 0,C 180,E1 -19925.27,E2 -19925.27} C_VEL
LIN {X 0,Y 227.931,Z 241.094,A -85,B 0,C 180,E1 -19927.328,E2 -19927.328} C_VEL
LIN {X 0,Y 227.792,Z 241.112,A -85,B 0,C 180,E1 -19932.741,E2 -19932.741} C_VEL
LIN {X 0,Y 227.79,Z 241.113,A -85,B 0,C 180,E1 -19937.252,E2 -19937.252} C_VEL
LIN {X 0,Y 227.828,Z 241.106,A -85,B 0,C 180,E1 -19941.905,E2 -19941.905} C_VEL
LIN {X 0,Y 227.856,Z 241.098,A -85,B 0,C 180,E1 -19946.376,E2 -19946.376} C_VEL
LIN {X 0,Y 227.861,Z 241.1,A -85,B 0,C 180,E1 -19950.429,E2 -19950.429} C_VEL
LIN {X 0,Y 227.893,Z 241.091,A -85,B 0,C 180,E1 -19954.421,E2 -19954.421} C_VEL
LIN {X 0,Y 227.894,Z 241.096,A -85,B 0,C 180,E1 -19958.28,E2 -19958.28} C_VEL
LIN {X 0,Y 227.992,Z 241.071,A -85,B 0,C 180,E1 -19963.892,E2 -19963.892} C_VEL
LIN {X 0,Y 228.027,Z 241.079,A -85,B 0,C 180,E1 -19967.54,E2 -19967.54} C_VEL
LIN {X 0,Y 228.224,Z 241.058,A -85,B 0,C 180,E1 -19971.142,E2 -19971.142} C_VEL
LIN {X 0,Y 228.287,Z 241.049,A -85,B 0,C 180,E1 -19972.926,E2 -19972.926} C_VEL
LIN {X 0,Y 228.518,Z 241.003,A -85,B 0,C 180,E1 -19978.237,E2 -19978.237} C_VEL
LIN {X 0,Y 228.52,Z 241.007,A -85,B 0,C 180,E1 -19981.762,E2 -19981.762} C_VEL
LIN {X 0,Y 228.289,Z 241.048,A -85,B 0,C 180,E1 -19987.073,E2 -19987.073} C_VEL
LIN {X 0,Y 228.114,Z 241.07,A -85,B 0,C 180,E1 -19990.652,E2 -19990.652} C_VEL
LIN {X 0,Y 228.018,Z 241.067,A -85,B 0,C 180,E1 -19996.104,E2 -19996.104} C_VEL
LIN {X 0,Y 227.941,Z 241.067,A -85,B 0,C 180,E1 -19999.825,E2 -19999.825} C_VEL
LIN {X 0,Y 227.915,Z 241.085,A -85,B 0,C 180,E1 -20003.632,E2 -20003.632} C_VEL
LIN {X 0,Y 227.864,Z 241.098,A -85,B 0,C 180,E1 -20007.557,E2 -20007.557} C_VEL
LIN {X 0,Y 227.848,Z 241.101,A -85,B 0,C 180,E1 -20011.625,E2 -20011.625} C_VEL
LIN {X 0,Y 227.864,Z 241.092,A -85,B 0,C 180,E1 -20015.874,E2 -20015.874} C_VEL
LIN {X 0,Y 227.873,Z 241.079,A -85,B 0,C 180,E1 -20020.366,E2 -20020.366} C_VEL
LIN {X 0,Y 227.889,Z 241.087,A -85,B 0,C 180,E1 -20022.723,E2 -20022.723} C_VEL
LIN {X 0,Y 227.799,Z 241.106,A -85,B 0,C 180,E1 -20027.261,E2 -20027.261} C_VEL
LIN {X 0,Y 227.831,Z 241.104,A -85,B 0,C 180,E1 -20031.912,E2 -20031.912} C_VEL
LIN {X 0,Y 227.869,Z 241.085,A -85,B 0,C 180,E1 -20036.38,E2 -20036.38} C_VEL
LIN {X 0,Y 227.911,Z 241.088,A -85,B 0,C 180,E1 -20040.441,E2 -20040.441} C_VEL
LIN {X 0,Y 227.922,Z 241.093,A -85,B 0,C 180,E1 -20044.428,E2 -20044.428} C_VEL
LIN {X 0,Y 227.957,Z 241.085,A -85,B 0,C 180,E1 -20048.289,E2 -20048.289} C_VEL
LIN {X 0,Y 228.031,Z 241.073,A -85,B 0,C 180,E1 -20052.828,E2 -20052.828} C_VEL
LIN {X 0,Y 228.091,Z 241.073,A -85,B 0,C 180,E1 -20057.546,E2 -20057.546} C_VEL
LIN {X 0,Y 228.303,Z 241.041,A -85,B 0,C 180,E1 -20061.147,E2 -20061.147} C_VEL
LIN {X 0,Y 228.352,Z 241.039,A -85,B 0,C 180,E1 -20062.929,E2 -20062.929} C_VEL
LIN {X 0,Y 228.553,Z 241.012,A -85,B 0,C 180,E1 -20068.238,E2 -20068.238} C_VEL
LIN {X 0,Y 228.553,Z 241.013,A -85,B 0,C 180,E1 -20071.762,E2 -20071.762} C_VEL
LIN {X 0,Y 228.339,Z 241.043,A -85,B 0,C 180,E1 -20077.071,E2 -20077.071} C_VEL
LIN {X 0,Y 228.143,Z 241.068,A -85,B 0,C 180,E1 -20080.65,E2 -20080.65} C_VEL
LIN {X 0,Y 228.061,Z 241.079,A -85,B 0,C 180,E1 -20084.271,E2 -20084.271} C_VEL
LIN {X 0,Y 227.998,Z 241.085,A -85,B 0,C 180,E1 -20088.765,E2 -20088.765} C_VEL
LIN {X 0,Y 229.526,Z 245.282,A -85,B 0,C 180,E1 -20089.134,E2 -20089.134} C_VEL
LIN {X 0,Y 237.452,Z 264.36,A -85,B 0,C 180,E1 -20090.688,E2 -20090.688} C_VEL
LIN {X 0,Y 241.443,Z 275.84,A -85,B 0,C 180,E1 -20091.503,E2 -20091.503} C_VEL
LIN {X 0,Y 238.486,Z 344.09,A -85,B 0,C 180,E1 -20093.896,E2 -20093.896} C_VEL
LIN {X 0,Y 237.516,Z 357.703,A -85,B 0,C 180,E1 -20094.703,E2 -20094.703} C_VEL
LIN {X 0,Y 236.445,Z 370.05,A -85,B 0,C 180,E1 -20095.764,E2 -20095.764} C_VEL
LIN {X 0,Y 234.93,Z 382.919,A -85,B 0,C 180,E1 -20097.26,E2 -20097.26} C_VEL
LIN {X 0,Y 233.525,Z 393.173,A -85,B 0,C 180,E1 -20098.782,E2 -20098.782} C_VEL
LIN {X 0,Y 231.913,Z 403.962,A -85,B 0,C 180,E1 -20100.776,E2 -20100.776} C_VEL
LIN {X 0,Y 230.367,Z 413.166,A -85,B 0,C 180,E1 -20102.9,E2 -20102.9} C_VEL
LIN {X 0,Y 228.904,Z 421.681,A -85,B 0,C 180,E1 -20105.322,E2 -20105.322} C_VEL
LIN {X 0,Y 227.621,Z 429.56,A -85,B 0,C 180,E1 -20108.13,E2 -20108.13} C_VEL
LIN {X 0,Y 226.655,Z 436.244,A -85,B 0,C 180,E1 -20111.232,E2 -20111.232} C_VEL
LIN {X 0,Y 225.984,Z 441.281,A -85,B 0,C 180,E1 -20114.334,E2 -20114.334} C_VEL
LIN {X 0,Y 225.592,Z 444.128,A -85,B 0,C 180,E1 -20116.735,E2 -20116.735} C_VEL
LIN {X 0,Y 225.468,Z 446.167,A -85,B 0,C 180,E1 -20119.113,E2 -20119.113} C_VEL
LIN {X 0,Y 225.557,Z 447.473,A -85,B 0,C 180,E1 -20121.453,E2 -20121.453} C_VEL
LIN {X 0,Y 225.839,Z 448.075,A -85,B 0,C 180,E1 -20124,E2 -20124} C_VEL
LIN {X 0,Y 226.534,Z 447.768,A -85,B 0,C 180,E1 -20126.883,E2 -20126.883} C_VEL
LIN {X 0,Y 227.648,Z 446.364,A -85,B 0,C 180,E1 -20129.806,E2 -20129.806} C_VEL
LIN {X 0,Y 229.184,Z 443.748,A -85,B 0,C 180,E1 -20132.773,E2 -20132.773} C_VEL
LIN {X 0,Y 231.221,Z 439.809,A -85,B 0,C 180,E1 -20135.749,E2 -20135.749} C_VEL
LIN {X 0,Y 233.995,Z 434.03,A -85,B 0,C 180,E1 -20138.875,E2 -20138.875} C_VEL
LIN {X 0,Y 237.009,Z 427.287,A -85,B 0,C 180,E1 -20141.584,E2 -20141.584} C_VEL
LIN {X 0,Y 239.729,Z 420.39,A -85,B 0,C 180,E1 -20143.783,E2 -20143.783} C_VEL
LIN {X 0,Y 242.959,Z 411.723,A -85,B 0,C 180,E1 -20145.981,E2 -20145.981} C_VEL
LIN {X 0,Y 246.276,Z 402.03,A -85,B 0,C 180,E1 -20147.931,E2 -20147.931} C_VEL
LIN {X 0,Y 249.298,Z 391.553,A -85,B 0,C 180,E1 -20149.607,E2 -20149.607} C_VEL
LIN {X 0,Y 251.97,Z 380.695,A -85,B 0,C 180,E1 -20150.974,E2 -20150.974} C_VEL
LIN {X 0,Y 254.457,Z 368.32,A -85,B 0,C 180,E1 -20152.174,E2 -20152.174} C_VEL
LIN {X 0,Y 256.272,Z 355.596,A -85,B 0,C 180,E1 -20153.087,E2 -20153.087} C_VEL
LIN {X 0,Y 257.666,Z 342.199,A -85,B 0,C 180,E1 -20153.708,E2 -20153.708} C_VEL
LIN {X 0,Y 261.307,Z 292.383,A -85,B 0,C 180,E1 -20155.403,E2 -20155.403} C_VEL
LIN {X 0,Y 256.543,Z 282.162,A -85,B 0,C 180,E1 -20157.165,E2 -20157.165} C_VEL
LIN {X 0,Y 252.432,Z 274.74,A -85,B 0,C 180,E1 -20158.762,E2 -20158.762} C_VEL
LIN {X 0,Y 246.487,Z 264.975,A -85,B 0,C 180,E1 -20161.292,E2 -20161.292} C_VEL
LIN {X 0,Y 243.601,Z 260.95,A -85,B 0,C 180,E1 -20162.627,E2 -20162.627} C_VEL
LIN {X 0,Y 240.771,Z 257.174,A -85,B 0,C 180,E1 -20164.041,E2 -20164.041} C_VEL
LIN {X 0,Y 238.216,Z 254.386,A -85,B 0,C 180,E1 -20165.397,E2 -20165.397} C_VEL
LIN {X 0,Y 236.515,Z 251.99,A -85,B 0,C 180,E1 -20166.398,E2 -20166.398} C_VEL
LIN {X 0,Y 233.967,Z 249.103,A -85,B 0,C 180,E1 -20168.01,E2 -20168.01} C_VEL
LIN {X 0,Y 233.048,Z 247.701,A -85,B 0,C 180,E1 -20168.673,E2 -20168.673} C_VEL
LIN {X 0,Y 229.004,Z 243.843,A -85,B 0,C 180,E1 -20171.788,E2 -20171.788} C_VEL
LIN {X 0,Y 228.448,Z 242.782,A -85,B 0,C 180,E1 -20172.437,E2 -20172.437} C_VEL
LIN {X 0,Y 227.993,Z 241.083,A -85,B 0,C 180,E1 -20176.108,E2 -20176.108} C_VEL
LIN {X 0,Y 227.855,Z 241.095,A -85,B 0,C 180,E1 -20180.921,E2 -20180.921} C_VEL
LIN {X 0,Y 227.34,Z 241.427,A -85,B 0,C 180,E1 -20182.397,E2 -20182.397} C_VEL
LIN {X 0,Y 225.04,Z 242.959,A -85,B 0,C 180,E1 -20184.804,E2 -20184.804} C_VEL
LIN {X 0,Y 222.479,Z 245.209,A -85,B 0,C 180,E1 -20187.755,E2 -20187.755} C_VEL
LIN {X 0,Y 222.279,Z 245.783,A -85,B 0,C 180,E1 -20188.772,E2 -20188.772} C_VEL
LIN {X 0,Y 222.967,Z 247.749,A -85,B 0,C 180,E1 -20192.266,E2 -20192.266} C_VEL
LIN {X 0,Y 224.65,Z 250.341,A -85,B 0,C 180,E1 -20194.68,E2 -20194.68} C_VEL
LIN {X 0,Y 229.003,Z 256.065,A -85,B 0,C 180,E1 -20198.983,E2 -20198.983} C_VEL
LIN {X 0,Y 233.877,Z 263.159,A -85,B 0,C 180,E1 -20202.553,E2 -20202.553} C_VEL
LIN {X 0,Y 238.12,Z 269.89,A -85,B 0,C 180,E1 -20205.102,E2 -20205.102} C_VEL
LIN {X 0,Y 241.949,Z 276.379,A -85,B 0,C 180,E1 -20207.122,E2 -20207.122} C_VEL
LIN {X 0,Y 244.832,Z 281.692,A -85,B 0,C 180,E1 -20208.532,E2 -20208.532} C_VEL
LIN {X 0,Y 248.755,Z 289.564,A -85,B 0,C 180,E1 -20210.295,E2 -20210.295} C_VEL
LIN {X 0,Y 253.152,Z 299.838,A -85,B 0,C 180,E1 -20212.179,E2 -20212.179} C_VEL
LIN {X 0,Y 253.874,Z 301.901,A -85,B 0,C 180,E1 -20212.486,E2 -20212.486} C_VEL
LIN {X 0,Y 255.097,Z 316.333,A -85,B 0,C 180,E1 -20213.589,E2 -20213.589} C_VEL
LIN {X 0,Y 251.372,Z 363.026,A -85,B 0,C 180,E1 -20215.219,E2 -20215.219} C_VEL
LIN {X 0,Y 249.56,Z 375.895,A -85,B 0,C 180,E1 -20215.908,E2 -20215.908} C_VEL
LIN {X 0,Y 247.099,Z 388.15,A -85,B 0,C 180,E1 -20216.808,E2 -20216.808} C_VEL
LIN {X 0,Y 244.02,Z 400.491,A -85,B 0,C 180,E1 -20218.051,E2 -20218.051} C_VEL
LIN {X 0,Y 240.725,Z 411.637,A -85,B 0,C 180,E1 -20219.522,E2 -20219.522} C_VEL
LIN {X 0,Y 237.379,Z 421.823,A -85,B 0,C 180,E1 -20221.245,E2 -20221.245} C_VEL
LIN {X 0,Y 233.95,Z 431.111,A -85,B 0,C 180,E1 -20223.22,E2 -20223.22} C_VEL
LIN {X 0,Y 230.742,Z 438.84,A -85,B 0,C 180,E1 -20225.244,E2 -20225.244} C_VEL
LIN {X 0,Y 227.065,Z 447.619,A -85,B 0,C 180,E1 -20228.199,E2 -20228.199} C_VEL
LIN {X 0,Y 224.538,Z 453.643,A -85,B 0,C 180,E1 -20230.815,E2 -20230.815} C_VEL
LIN {X 0,Y 222.285,Z 458.457,A -85,B 0,C 180,E1 -20233.47,E2 -20233.47} C_VEL
LIN {X 0,Y 220.567,Z 462.179,A -85,B 0,C 180,E1 -20236.175,E2 -20236.175} C_VEL
LIN {X 0,Y 219.513,Z 464.915,A -85,B 0,C 180,E1 -20238.926,E2 -20238.926} C_VEL
LIN {X 0,Y 219.011,Z 466.25,A -85,B 0,C 180,E1 -20240.768,E2 -20240.768} C_VEL
LIN {X 0,Y 218.691,Z 467.153,A -85,B 0,C 180,E1 -20242.615,E2 -20242.615} C_VEL
LIN {X 0,Y 218.55,Z 467.781,A -85,B 0,C 180,E1 -20245.479,E2 -20245.479} C_VEL
LIN {X 0,Y 218.753,Z 467.477,A -85,B 0,C 180,E1 -20248.159,E2 -20248.159} C_VEL
LIN {X 0,Y 218.812,Z 466.753,A -85,B 0,C 180,E1 -20250,E2 -20250} C_VEL
LIN {X 0,Y 218.799,Z 465.574,A -85,B 0,C 180,E1 -20251.84,E2 -20251.84} C_VEL
LIN {X 0,Y 218.762,Z 463.961,A -85,B 0,C 180,E1 -20253.683,E2 -20253.683} C_VEL
LIN {X 0,Y 218.827,Z 460.644,A -85,B 0,C 180,E1 -20256.453,E2 -20256.453} C_VEL
LIN {X 0,Y 219.08,Z 456.174,A -85,B 0,C 180,E1 -20259.229,E2 -20259.229} C_VEL
LIN {X 0,Y 219.667,Z 450.432,A -85,B 0,C 180,E1 -20262.001,E2 -20262.001} C_VEL
LIN {X 0,Y 220.796,Z 443.195,A -85,B 0,C 180,E1 -20264.751,E2 -20264.751} C_VEL
LIN {X 0,Y 222.246,Z 434.105,A -85,B 0,C 180,E1 -20267.48,E2 -20267.48} C_VEL
LIN {X 0,Y 223.554,Z 426.162,A -85,B 0,C 180,E1 -20269.415,E2 -20269.415} C_VEL
LIN {X 0,Y 225.232,Z 415.651,A -85,B 0,C 180,E1 -20271.506,E2 -20271.506} C_VEL
LIN {X 0,Y 226.963,Z 404.475,A -85,B 0,C 180,E1 -20273.251,E2 -20273.251} C_VEL
LIN {X 0,Y 228.837,Z 392.158,A -85,B 0,C 180,E1 -20274.733,E2 -20274.733} C_VEL
LIN {X 0,Y 230.135,Z 380.532,A -85,B 0,C 180,E1 -20275.793,E2 -20275.793} C_VEL
LIN {X 0,Y 231.389,Z 366.451,A -85,B 0,C 180,E1 -20276.673,E2 -20276.673} C_VEL
LIN {X 0,Y 233.053,Z 327.718,A -85,B 0,C 180,E1 -20278.121,E2 -20278.121} C_VEL
LIN {X 0,Y 233.638,Z 309.518,A -85,B 0,C 180,E1 -20278.787,E2 -20278.787} C_VEL
LIN {X 0,Y 229.184,Z 271.739,A -85,B 0,C 180,E1 -20280.74,E2 -20280.74} C_VEL
LIN {X 0,Y 223.846,Z 256.279,A -85,B 0,C 180,E1 -20281.93,E2 -20281.93} C_VEL
LIN {X 0,Y 221.897,Z 246.604,A -85,B 0,C 180,E1 -20285.863,E2 -20285.863} C_VEL
LIN {X 0,Y 220.886,Z 241.972,A -85,B 0,C 180,E1 -20287.907,E2 -20287.907} C_VEL
LIN {X 0,Y 220.748,Z 241.989,A -85,B 0,C 180,E1 -20292.923,E2 -20292.923} C_VEL
LIN {X 0,Y 220.746,Z 241.99,A -85,B 0,C 180,E1 -20297.069,E2 -20297.069} C_VEL
LIN {X 0,Y 220.77,Z 241.984,A -85,B 0,C 180,E1 -20300.454,E2 -20300.454} C_VEL
LIN {X 0,Y 220.81,Z 241.978,A -85,B 0,C 180,E1 -20302.789,E2 -20302.789} C_VEL
LIN {X 0,Y 220.787,Z 241.98,A -85,B 0,C 180,E1 -20307.238,E2 -20307.238} C_VEL
LIN {X 0,Y 220.79,Z 241.981,A -85,B 0,C 180,E1 -20311.479,E2 -20311.479} C_VEL
LIN {X 0,Y 220.832,Z 241.975,A -85,B 0,C 180,E1 -20315.56,E2 -20315.56} C_VEL
LIN {X 0,Y 220.826,Z 241.978,A -85,B 0,C 180,E1 -20319.507,E2 -20319.507} C_VEL
LIN {X 0,Y 220.951,Z 241.95,A -85,B 0,C 180,E1 -20323.364,E2 -20323.364} C_VEL
LIN {X 0,Y 221.036,Z 241.951,A -85,B 0,C 180,E1 -20329.001,E2 -20329.001} C_VEL
LIN {X 0,Y 221.222,Z 241.928,A -85,B 0,C 180,E1 -20332.699,E2 -20332.699} C_VEL
LIN {X 0,Y 221.452,Z 241.882,A -85,B 0,C 180,E1 -20338.181,E2 -20338.181} C_VEL
LIN {X 0,Y 221.478,Z 241.884,A -85,B 0,C 180,E1 -20341.818,E2 -20341.818} C_VEL
LIN {X 0,Y 221.224,Z 241.927,A -85,B 0,C 180,E1 -20347.3,E2 -20347.3} C_VEL
LIN {X 0,Y 221.035,Z 241.949,A -85,B 0,C 180,E1 -20350.997,E2 -20350.997} C_VEL
LIN {X 0,Y 220.983,Z 241.937,A -85,B 0,C 180,E1 -20356.632,E2 -20356.632} C_VEL
LIN {X 0,Y 220.898,Z 241.946,A -85,B 0,C 180,E1 -20360.485,E2 -20360.485} C_VEL
LIN {X 0,Y 220.859,Z 241.967,A -85,B 0,C 180,E1 -20364.435,E2 -20364.435} C_VEL
LIN {X 0,Y 220.815,Z 241.98,A -85,B 0,C 180,E1 -20368.516,E2 -20368.516} C_VEL
LIN {X 0,Y 220.797,Z 241.977,A -85,B 0,C 180,E1 -20372.759,E2 -20372.759} C_VEL
LIN {X 0,Y 220.821,Z 241.961,A -85,B 0,C 180,E1 -20377.29,E2 -20377.29} C_VEL
LIN {X 0,Y 220.834,Z 241.959,A -85,B 0,C 180,E1 -20381.937,E2 -20381.937} C_VEL
LIN {X 0,Y 220.768,Z 241.979,A -85,B 0,C 180,E1 -20385.551,E2 -20385.551} C_VEL
LIN {X 0,Y 220.794,Z 241.98,A -85,B 0,C 180,E1 -20390.466,E2 -20390.466} C_VEL
LIN {X 0,Y 220.791,Z 241.972,A -85,B 0,C 180,E1 -20395.048,E2 -20395.048} C_VEL
LIN {X 0,Y 220.86,Z 241.96,A -85,B 0,C 180,E1 -20399.398,E2 -20399.398} C_VEL
LIN {X 0,Y 220.889,Z 241.97,A -85,B 0,C 180,E1 -20403.552,E2 -20403.552} C_VEL
LIN {X 0,Y 220.872,Z 241.972,A -85,B 0,C 180,E1 -20407.556,E2 -20407.556} C_VEL
LIN {X 0,Y 220.98,Z 241.951,A -85,B 0,C 180,E1 -20412.573,E2 -20412.573} C_VEL
LIN {X 0,Y 221.023,Z 241.954,A -85,B 0,C 180,E1 -20417.141,E2 -20417.141} C_VEL
LIN {X 0,Y 221.234,Z 241.92,A -85,B 0,C 180,E1 -20420.862,E2 -20420.862} C_VEL
LIN {X 0,Y 221.287,Z 241.919,A -85,B 0,C 180,E1 -20422.702,E2 -20422.702} C_VEL
LIN {X 0,Y 221.511,Z 241.889,A -85,B 0,C 180,E1 -20428.182,E2 -20428.182} C_VEL
LIN {X 0,Y 221.511,Z 241.89,A -85,B 0,C 180,E1 -20431.818,E2 -20431.818} C_VEL
LIN {X 0,Y 221.271,Z 241.925,A -85,B 0,C 180,E1 -20437.298,E2 -20437.298} C_VEL
LIN {X 0,Y 221.079,Z 241.951,A -85,B 0,C 180,E1 -20440.995,E2 -20440.995} C_VEL
LIN {X 0,Y 221.028,Z 241.954,A -85,B 0,C 180,E1 -20446.627,E2 -20446.627} C_VEL
LIN {X 0,Y 220.978,Z 242.055,A -85,B 0,C 180,E1 -20448.079,E2 -20448.079} C_VEL
LIN {X 0,Y 222.55,Z 246.325,A -85,B 0,C 180,E1 -20448.437,E2 -20448.437} C_VEL
LIN {X 0,Y 231.308,Z 267.303,A -85,B 0,C 180,E1 -20450.208,E2 -20450.208} C_VEL
LIN {X 0,Y 234.755,Z 277.225,A -85,B 0,C 180,E1 -20450.937,E2 -20450.937} C_VEL
LIN {X 0,Y 231.655,Z 345.149,A -85,B 0,C 180,E1 -20453.396,E2 -20453.396} C_VEL
LIN {X 0,Y 230.697,Z 359.129,A -85,B 0,C 180,E1 -20454.277,E2 -20454.277} C_VEL
LIN {X 0,Y 229.552,Z 371.237,A -85,B 0,C 180,E1 -20455.378,E2 -20455.378} C_VEL
LIN {X 0,Y 228.054,Z 383.284,A -85,B 0,C 180,E1 -20456.83,E2 -20456.83} C_VEL
LIN {X 0,Y 226.531,Z 394.056,A -85,B 0,C 180,E1 -20458.486,E2 -20458.486} C_VEL
LIN {X 0,Y 224.87,Z 404.611,A -85,B 0,C 180,E1 -20460.518,E2 -20460.518} C_VEL
LIN {X 0,Y 223.201,Z 414.449,A -85,B 0,C 180,E1 -20462.895,E2 -20462.895} C_VEL
LIN {X 0,Y 221.752,Z 422.613,A -85,B 0,C 180,E1 -20465.334,E2 -20465.334} C_VEL
LIN {X 0,Y 220.618,Z 429.354,A -85,B 0,C 180,E1 -20467.817,E2 -20467.817} C_VEL
LIN {X 0,Y 219.72,Z 435.018,A -85,B 0,C 180,E1 -20470.403,E2 -20470.403} C_VEL
LIN {X 0,Y 219.275,Z 438.742,A -85,B 0,C 180,E1 -20472.51,E2 -20472.51} C_VEL
LIN {X 0,Y 218.741,Z 442.337,A -85,B 0,C 180,E1 -20475.022,E2 -20475.022} C_VEL
LIN {X 0,Y 218.424,Z 445.225,A -85,B 0,C 180,E1 -20477.729,E2 -20477.729} C_VEL
LIN {X 0,Y 218.375,Z 447.24,A -85,B 0,C 180,E1 -20480.562,E2 -20480.562} C_VEL
LIN {X 0,Y 218.649,Z 448.293,A -85,B 0,C 180,E1 -20483.464,E2 -20483.464} C_VEL
LIN {X 0,Y 219.495,Z 448.202,A -85,B 0,C 180,E1 -20487.022,E2 -20487.022} C_VEL
LIN {X 0,Y 220.373,Z 447.294,A -85,B 0,C 180,E1 -20489.426,E2 -20489.426} C_VEL
LIN {X 0,Y 221.873,Z 445.097,A -85,B 0,C 180,E1 -20492.477,E2 -20492.477} C_VEL
LIN {X 0,Y 224.224,Z 441.066,A -85,B 0,C 180,E1 -20495.955,E2 -20495.955} C_VEL
LIN {X 0,Y 226.487,Z 436.767,A -85,B 0,C 180,E1 -20498.562,E2 -20498.562} C_VEL
LIN {X 0,Y 229.673,Z 430.249,A -85,B 0,C 180,E1 -20501.532,E2 -20501.532} C_VEL
LIN {X 0,Y 233.108,Z 422.485,A -85,B 0,C 180,E1 -20504.256,E2 -20504.256} C_VEL
LIN {X 0,Y 236.473,Z 414.143,A -85,B 0,C 180,E1 -20506.54,E2 -20506.54} C_VEL
LIN {X 0,Y 239.978,Z 404.521,A -85,B 0,C 180,E1 -20508.599,E2 -20508.599} C_VEL
LIN {X 0,Y 243.374,Z 393.837,A -85,B 0,C 180,E1 -20510.406,E2 -20510.406} C_VEL
LIN {X 0,Y 246.42,Z 382.273,A -85,B 0,C 180,E1 -20511.934,E2 -20511.934} C_VEL
LIN {X 0,Y 249.109,Z 369.864,A -85,B 0,C 180,E1 -20513.187,E2 -20513.187} C_VEL
LIN {X 0,Y 251.146,Z 357.053,A -85,B 0,C 180,E1 -20514.153,E2 -20514.153} C_VEL
LIN {X 0,Y 252.616,Z 344.165,A -85,B 0,C 180,E1 -20514.788,E2 -20514.788} C_VEL
LIN {X 0,Y 256.43,Z 295.121,A -85,B 0,C 180,E1 -20516.483,E2 -20516.483} C_VEL
LIN {X 0,Y 251.755,Z 285.111,A -85,B 0,C 180,E1 -20518.345,E2 -20518.345} C_VEL
LIN {X 0,Y 246.654,Z 276.066,A -85,B 0,C 180,E1 -20520.49,E2 -20520.49} C_VEL
LIN {X 0,Y 242.965,Z 269.976,A -85,B 0,C 180,E1 -20522.223,E2 -20522.223} C_VEL
LIN {X 0,Y 240.807,Z 266.866,A -85,B 0,C 180,E1 -20523.278,E2 -20523.278} C_VEL
LIN {X 0,Y 238.296,Z 263.464,A -85,B 0,C 180,E1 -20524.609,E2 -20524.609} C_VEL
LIN {X 0,Y 235.529,Z 260.184,A -85,B 0,C 180,E1 -20526.157,E2 -20526.157} C_VEL
LIN {X 0,Y 234.231,Z 258.307,A -85,B 0,C 180,E1 -20526.982,E2 -20526.982} C_VEL
LIN {X 0,Y 231.693,Z 255.26,A -85,B 0,C 180,E1 -20528.683,E2 -20528.683} C_VEL
LIN {X 0,Y 230.574,Z 253.72,A -85,B 0,C 180,E1 -20529.525,E2 -20529.525} C_VEL
LIN {X 0,Y 227.306,Z 250.565,A -85,B 0,C 180,E1 -20532.203,E2 -20532.203} C_VEL
LIN {X 0,Y 226.532,Z 249.375,A -85,B 0,C 180,E1 -20532.999,E2 -20532.999} C_VEL
LIN {X 0,Y 223.579,Z 246.646,A -85,B 0,C 180,E1 -20536.434,E2 -20536.434} C_VEL
LIN {X 0,Y 221.706,Z 244.629,A -85,B 0,C 180,E1 -20540.142,E2 -20540.142} C_VEL
LIN {X 0,Y 221.739,Z 244.666,A -85,B 0,C 180,E1 -20544.333,E2 -20544.333} C_VEL
LIN {X 0,Y 222.259,Z 245.566,A -85,B 0,C 180,E1 -20548.315,E2 -20548.315} C_VEL
LIN {X 0,Y 222.279,Z 245.783,A -85,B 0,C 180,E1 -20548.772,E2 -20548.772} C_VEL
LIN {X 0,Y 222.363,Z 247.279,A -85,B 0,C 180,E1 -20550.245,E2 -20550.245} C_VEL
LIN {X 0,Y 222.491,Z 249.873,A -85,B 0,C 180,E1 -20551.628,E2 -20551.628} C_VEL
LIN {X 0,Y 223.28,Z 256.146,A -85,B 0,C 180,E1 -20554.271,E2 -20554.271} C_VEL
LIN {X 0,Y 224.2,Z 258.779,A -85,B 0,C 180,E1 -20555.636,E2 -20555.636} C_VEL
LIN {X 0,Y 224.622,Z 259.444,A -85,B 0,C 180,E1 -20556.108,E2 -20556.108} C_VEL
LIN {X 0,Y 227.015,Z 262.505,A -85,B 0,C 180,E1 -20558.397,E2 -20558.397} C_VEL
LIN {X 0,Y 231.572,Z 269.45,A -85,B 0,C 180,E1 -20561.936,E2 -20561.936} C_VEL
LIN {X 0,Y 235.44,Z 275.846,A -85,B 0,C 180,E1 -20564.4,E2 -20564.4} C_VEL
LIN {X 0,Y 239.018,Z 282.164,A -85,B 0,C 180,E1 -20566.422,E2 -20566.422} C_VEL
LIN {X 0,Y 241.854,Z 287.6,A -85,B 0,C 180,E1 -20567.875,E2 -20567.875} C_VEL
LIN {X 0,Y 245.94,Z 296.292,A -85,B 0,C 180,E1 -20569.834,E2 -20569.834} C_VEL
LIN {X 0,Y 249.422,Z 305.127,A -85,B 0,C 180,E1 -20571.434,E2 -20571.434} C_VEL
LIN {X 0,Y 250.35,Z 318.07,A -85,B 0,C 180,E1 -20572.451,E2 -20572.451} C_VEL
LIN {X 0,Y 246.558,Z 362.675,A -85,B 0,C 180,E1 -20574.006,E2 -20574.006} C_VEL
LIN {X 0,Y 244.582,Z 376.122,A -85,B 0,C 180,E1 -20574.739,E2 -20574.739} C_VEL
LIN {X 0,Y 241.787,Z 389.142,A -85,B 0,C 180,E1 -20575.729,E2 -20575.729} C_VEL
LIN {X 0,Y 238.571,Z 401.109,A -85,B 0,C 180,E1 -20576.98,E2 -20576.98} C_VEL
LIN {X 0,Y 235.136,Z 412.014,A -85,B 0,C 180,E1 -20578.466,E2 -20578.466} C_VEL
LIN {X 0,Y 231.26,Z 423.002,A -85,B 0,C 180,E1 -20580.41,E2 -20580.41} C_VEL
LIN {X 0,Y 227.7,Z 432.014,A -85,B 0,C 180,E1 -20582.424,E2 -20582.424} C_VEL
LIN {X 0,Y 224.359,Z 439.544,A -85,B 0,C 180,E1 -20584.49,E2 -20584.49} C_VEL
LIN {X 0,Y 220.996,Z 446.99,A -85,B 0,C 180,E1 -20587.075,E2 -20587.075} C_VEL
LIN {X 0,Y 218.599,Z 452.103,A -85,B 0,C 180,E1 -20589.291,E2 -20589.291} C_VEL
LIN {X 0,Y 216.238,Z 457.137,A -85,B 0,C 180,E1 -20592.017,E2 -20592.017} C_VEL
LIN {X 0,Y 214.177,Z 461.094,A -85,B 0,C 180,E1 -20594.782,E2 -20594.782} C_VEL
LIN {X 0,Y 212.503,Z 464.837,A -85,B 0,C 180,E1 -20598.556,E2 -20598.556} C_VEL
LIN {X 0,Y 211.993,Z 466.071,A -85,B 0,C 180,E1 -20600.46,E2 -20600.46} C_VEL
LIN {X 0,Y 211.489,Z 467.339,A -85,B 0,C 180,E1 -20604.279,E2 -20604.279} C_VEL
LIN {X 0,Y 211.487,Z 467.395,A -85,B 0,C 180,E1 -20606.189,E2 -20606.189} C_VEL
LIN {X 0,Y 211.68,Z 467.042,A -85,B 0,C 180,E1 -20608.097,E2 -20608.097} C_VEL
LIN {X 0,Y 211.744,Z 466.232,A -85,B 0,C 180,E1 -20610,E2 -20610} C_VEL
LIN {X 0,Y 211.732,Z 464.998,A -85,B 0,C 180,E1 -20611.902,E2 -20611.902} C_VEL
LIN {X 0,Y 211.716,Z 461.783,A -85,B 0,C 180,E1 -20615.207,E2 -20615.207} C_VEL
LIN {X 0,Y 211.895,Z 456.939,A -85,B 0,C 180,E1 -20618.582,E2 -20618.582} C_VEL
LIN {X 0,Y 212.438,Z 451.478,A -85,B 0,C 180,E1 -20621.448,E2 -20621.448} C_VEL
LIN {X 0,Y 213.43,Z 444.596,A -85,B 0,C 180,E1 -20624.296,E2 -20624.296} C_VEL
LIN {X 0,Y 214.811,Z 435.982,A -85,B 0,C 180,E1 -20627.123,E2 -20627.123} C_VEL
LIN {X 0,Y 216.452,Z 426.518,A -85,B 0,C 180,E1 -20629.58,E2 -20629.58} C_VEL
LIN {X 0,Y 218.169,Z 416.156,A -85,B 0,C 180,E1 -20631.741,E2 -20631.741} C_VEL
LIN {X 0,Y 219.727,Z 406.76,A -85,B 0,C 180,E1 -20633.314,E2 -20633.314} C_VEL
LIN {X 0,Y 221.531,Z 395.139,A -85,B 0,C 180,E1 -20634.854,E2 -20634.854} C_VEL
LIN {X 0,Y 223.138,Z 382.034,A -85,B 0,C 180,E1 -20636.161,E2 -20636.161} C_VEL
LIN {X 0,Y 224.399,Z 369.081,A -85,B 0,C 180,E1 -20637.068,E2 -20637.068} C_VEL
LIN {X 0,Y 225.305,Z 352.917,A -85,B 0,C 180,E1 -20637.768,E2 -20637.768} C_VEL
LIN {X 0,Y 227.003,Z 310.486,A -85,B 0,C 180,E1 -20639.355,E2 -20639.355} C_VEL
LIN {X 0,Y 222.762,Z 273.973,A -85,B 0,C 180,E1 -20641.288,E2 -20641.288} C_VEL
LIN {X 0,Y 216.565,Z 255.923,A -85,B 0,C 180,E1 -20642.754,E2 -20642.754} C_VEL
LIN {X 0,Y 214.332,Z 245.142,A -85,B 0,C 180,E1 -20647.323,E2 -20647.323} C_VEL
LIN {X 0,Y 213.807,Z 242.853,A -85,B 0,C 180,E1 -20648.423,E2 -20648.423} C_VEL
LIN {X 0,Y 213.693,Z 242.87,A -85,B 0,C 180,E1 -20653.676,E2 -20653.676} C_VEL
LIN {X 0,Y 213.691,Z 242.869,A -85,B 0,C 180,E1 -20656.341,E2 -20656.341} C_VEL
LIN {X 0,Y 213.695,Z 242.867,A -85,B 0,C 180,E1 -20659.142,E2 -20659.142} C_VEL
LIN {X 0,Y 213.728,Z 242.862,A -85,B 0,C 180,E1 -20663.708,E2 -20663.708} C_VEL
LIN {X 0,Y 213.739,Z 242.86,A -85,B 0,C 180,E1 -20668.257,E2 -20668.257} C_VEL
LIN {X 0,Y 213.791,Z 242.849,A -85,B 0,C 180,E1 -20672.598,E2 -20672.598} C_VEL
LIN {X 0,Y 213.778,Z 242.854,A -85,B 0,C 180,E1 -20676.985,E2 -20676.985} C_VEL
LIN {X 0,Y 213.86,Z 242.838,A -85,B 0,C 180,E1 -20682.796,E2 -20682.796} C_VEL
LIN {X 0,Y 213.905,Z 242.832,A -85,B 0,C 180,E1 -20686.703,E2 -20686.703} C_VEL
LIN {X 0,Y 214.101,Z 242.815,A -85,B 0,C 180,E1 -20690.553,E2 -20690.553} C_VEL
LIN {X 0,Y 214.06,Z 242.816,A -85,B 0,C 180,E1 -20694.347,E2 -20694.347} C_VEL
LIN {X 0,Y 214.389,Z 242.761,A -85,B 0,C 180,E1 -20698.121,E2 -20698.121} C_VEL
LIN {X 0,Y 214.507,Z 242.744,A -85,B 0,C 180,E1 -20699.999,E2 -20699.999} C_VEL
LIN {X 0,Y 214.411,Z 242.763,A -85,B 0,C 180,E1 -20701.878,E2 -20701.878} C_VEL
LIN {X 0,Y 214.162,Z 242.806,A -85,B 0,C 180,E1 -20707.542,E2 -20707.542} C_VEL
LIN {X 0,Y 213.967,Z 242.827,A -85,B 0,C 180,E1 -20711.365,E2 -20711.365} C_VEL
LIN {X 0,Y 213.89,Z 242.825,A -85,B 0,C 180,E1 -20715.239,E2 -20715.239} C_VEL
LIN {X 0,Y 213.858,Z 242.818,A -85,B 0,C 180,E1 -20719.185,E2 -20719.185} C_VEL
LIN {X 0,Y 213.84,Z 242.837,A -85,B 0,C 180,E1 -20723.227,E2 -20723.227} C_VEL
LIN {X 0,Y 213.809,Z 242.849,A -85,B 0,C 180,E1 -20727.452,E2 -20727.452} C_VEL
LIN {X 0,Y 213.748,Z 242.857,A -85,B 0,C 180,E1 -20731.74,E2 -20731.74} C_VEL
LIN {X 0,Y 213.726,Z 242.847,A -85,B 0,C 180,E1 -20736.291,E2 -20736.291} C_VEL
LIN {X 0,Y 213.778,Z 242.835,A -85,B 0,C 180,E1 -20740.883,E2 -20740.883} C_VEL
LIN {X 0,Y 213.764,Z 242.846,A -85,B 0,C 180,E1 -20743.679,E2 -20743.679} C_VEL
LIN {X 0,Y 213.699,Z 242.864,A -85,B 0,C 180,E1 -20748.878,E2 -20748.878} C_VEL
LIN {X 0,Y 213.733,Z 242.856,A -85,B 0,C 180,E1 -20753.714,E2 -20753.714} C_VEL
LIN {X 0,Y 213.772,Z 242.841,A -85,B 0,C 180,E1 -20758.734,E2 -20758.734} C_VEL
LIN {X 0,Y 213.819,Z 242.848,A -85,B 0,C 180,E1 -20762.606,E2 -20762.606} C_VEL
LIN {X 0,Y 213.847,Z 242.846,A -85,B 0,C 180,E1 -20766.955,E2 -20766.955} C_VEL
LIN {X 0,Y 213.94,Z 242.828,A -85,B 0,C 180,E1 -20772.805,E2 -20772.805} C_VEL
LIN {X 0,Y 213.978,Z 242.83,A -85,B 0,C 180,E1 -20776.71,E2 -20776.71} C_VEL
LIN {X 0,Y 214.165,Z 242.799,A -85,B 0,C 180,E1 -20780.557,E2 -20780.557} C_VEL
LIN {X 0,Y 214.225,Z 242.798,A -85,B 0,C 180,E1 -20782.461,E2 -20782.461} C_VEL
LIN {X 0,Y 214.444,Z 242.769,A -85,B 0,C 180,E1 -20788.122,E2 -20788.122} C_VEL
LIN {X 0,Y 214.549,Z 242.759,A -85,B 0,C 180,E1 -20790,E2 -20790} C_VEL
LIN {X 0,Y 214.444,Z 242.77,A -85,B 0,C 180,E1 -20791.878,E2 -20791.878} C_VEL
LIN {X 0,Y 214.208,Z 242.804,A -85,B 0,C 180,E1 -20797.54,E2 -20797.54} C_VEL
LIN {X 0,Y 214.006,Z 242.831,A -85,B 0,C 180,E1 -20801.363,E2 -20801.363} C_VEL
LIN {X 0,Y 213.936,Z 242.839,A -85,B 0,C 180,E1 -20805.235,E2 -20805.235} C_VEL
LIN {X 0,Y 213.983,Z 242.934,A -85,B 0,C 180,E1 -20807.321,E2 -20807.321} C_VEL
LIN {X 0,Y 216.006,Z 248.186,A -85,B 0,C 180,E1 -20807.784,E2 -20807.784} C_VEL
LIN {X 0,Y 225.24,Z 270.528,A -85,B 0,C 180,E1 -20809.745,E2 -20809.745} C_VEL
LIN {X 0,Y 228.107,Z 279.025,A -85,B 0,C 180,E1 -20810.378,E2 -20810.378} C_VEL
LIN {X 0,Y 224.988,Z 344.534,A -85,B 0,C 180,E1 -20812.814,E2 -20812.814} C_VEL
LIN {X 0,Y 223.995,Z 358.175,A -85,B 0,C 180,E1 -20813.67,E2 -20813.67} C_VEL
LIN {X 0,Y 222.747,Z 371.213,A -85,B 0,C 180,E1 -20814.861,E2 -20814.861} C_VEL
LIN {X 0,Y 221.156,Z 383.737,A -85,B 0,C 180,E1 -20816.414,E2 -20816.414} C_VEL
LIN {X 0,Y 219.466,Z 395.352,A -85,B 0,C 180,E1 -20818.27,E2 -20818.27} C_VEL
LIN {X 0,Y 217.78,Z 405.601,A -85,B 0,C 180,E1 -20820.346,E2 -20820.346} C_VEL
LIN {X 0,Y 215.999,Z 415.867,A -85,B 0,C 180,E1 -20822.945,E2 -20822.945} C_VEL
LIN {X 0,Y 214.496,Z 424.139,A -85,B 0,C 180,E1 -20825.576,E2 -20825.576} C_VEL
LIN {X 0,Y 213.122,Z 432.091,A -85,B 0,C 180,E1 -20828.791,E2 -20828.791} C_VEL
LIN {X 0,Y 212.409,Z 437.209,A -85,B 0,C 180,E1 -20831.427,E2 -20831.427} C_VEL
LIN {X 0,Y 211.796,Z 441.412,A -85,B 0,C 180,E1 -20834.168,E2 -20834.168} C_VEL
LIN {X 0,Y 211.397,Z 444.683,A -85,B 0,C 180,E1 -20836.997,E2 -20836.997} C_VEL
LIN {X 0,Y 211.288,Z 447.546,A -85,B 0,C 180,E1 -20840.804,E2 -20840.804} C_VEL
LIN {X 0,Y 211.546,Z 448.509,A -85,B 0,C 180,E1 -20843.274,E2 -20843.274} C_VEL
LIN {X 0,Y 212.075,Z 448.78,A -85,B 0,C 180,E1 -20845.934,E2 -20845.934} C_VEL
LIN {X 0,Y 213.086,Z 448.117,A -85,B 0,C 180,E1 -20849.03,E2 -20849.03} C_VEL
LIN {X 0,Y 214.9,Z 445.878,A -85,B 0,C 180,E1 -20852.752,E2 -20852.752} C_VEL
LIN {X 0,Y 217.301,Z 442.095,A -85,B 0,C 180,E1 -20856.277,E2 -20856.277} C_VEL
LIN {X 0,Y 220.149,Z 437.189,A -85,B 0,C 180,E1 -20859.442,E2 -20859.442} C_VEL
LIN {X 0,Y 223.107,Z 431.63,A -85,B 0,C 180,E1 -20862.114,E2 -20862.114} C_VEL
LIN {X 0,Y 226.092,Z 425.404,A -85,B 0,C 180,E1 -20864.476,E2 -20864.476} C_VEL
LIN {X 0,Y 229.193,Z 418.267,A -85,B 0,C 180,E1 -20866.657,E2 -20866.657} C_VEL
LIN {X 0,Y 233.023,Z 408.826,A -85,B 0,C 180,E1 -20868.915,E2 -20868.915} C_VEL
LIN {X 0,Y 236.826,Z 398.255,A -85,B 0,C 180,E1 -20870.911,E2 -20870.911} C_VEL
LIN {X 0,Y 240.21,Z 386.837,A -85,B 0,C 180,E1 -20872.592,E2 -20872.592} C_VEL
LIN {X 0,Y 243.054,Z 375.455,A -85,B 0,C 180,E1 -20873.88,E2 -20873.88} C_VEL
LIN {X 0,Y 245.531,Z 362.45,A -85,B 0,C 180,E1 -20874.997,E2 -20874.997} C_VEL
LIN {X 0,Y 247.316,Z 348.971,A -85,B 0,C 180,E1 -20875.806,E2 -20875.806} C_VEL
LIN {X 0,Y 251.607,Z 297.82,A -85,B 0,C 180,E1 -20877.631,E2 -20877.631} C_VEL
LIN {X 0,Y 247.216,Z 288.28,A -85,B 0,C 180,E1 -20879.532,E2 -20879.532} C_VEL
LIN {X 0,Y 240.859,Z 276.934,A -85,B 0,C 180,E1 -20882.519,E2 -20882.519} C_VEL
LIN {X 0,Y 238.236,Z 273.018,A -85,B 0,C 180,E1 -20883.865,E2 -20883.865} C_VEL
LIN {X 0,Y 235.969,Z 269.84,A -85,B 0,C 180,E1 -20885.127,E2 -20885.127} C_VEL
LIN {X 0,Y 233.104,Z 266.264,A -85,B 0,C 180,E1 -20886.819,E2 -20886.819} C_VEL
LIN {X 0,Y 231.899,Z 264.597,A -85,B 0,C 180,E1 -20887.623,E2 -20887.623} C_VEL
LIN {X 0,Y 229.402,Z 261.294,A -85,B 0,C 180,E1 -20889.418,E2 -20889.418} C_VEL
LIN {X 0,Y 227.809,Z 259.551,A -85,B 0,C 180,E1 -20890.668,E2 -20890.668} C_VEL
LIN {X 0,Y 225.479,Z 257.042,A -85,B 0,C 180,E1 -20892.775,E2 -20892.775} C_VEL
LIN {X 0,Y 224.538,Z 255.842,A -85,B 0,C 180,E1 -20893.768,E2 -20893.768} C_VEL
LIN {X 0,Y 222.144,Z 253.497,A -85,B 0,C 180,E1 -20896.791,E2 -20896.791} C_VEL
LIN {X 0,Y 220.318,Z 251.552,A -85,B 0,C 180,E1 -20900.543,E2 -20900.543} C_VEL
LIN {X 0,Y 219.523,Z 251.438,A -85,B 0,C 180,E1 -20904.595,E2 -20904.595} C_VEL
LIN {X 0,Y 220.029,Z 252.343,A -85,B 0,C 180,E1 -20908.292,E2 -20908.292} C_VEL
LIN {X 0,Y 221.652,Z 254.729,A -85,B 0,C 180,E1 -20912.075,E2 -20912.075} C_VEL
LIN {X 0,Y 223.379,Z 257.526,A -85,B 0,C 180,E1 -20914.632,E2 -20914.632} C_VEL
LIN {X 0,Y 224.622,Z 259.444,A -85,B 0,C 180,E1 -20916.108,E2 -20916.108} C_VEL
LIN {X 0,Y 225.82,Z 261.953,A -85,B 0,C 180,E1 -20917.428,E2 -20917.428} C_VEL
LIN {X 0,Y 226.811,Z 265.509,A -85,B 0,C 180,E1 -20918.608,E2 -20918.608} C_VEL
LIN {X 0,Y 228.786,Z 273.669,A -85,B 0,C 180,E1 -20920.787,E2 -20920.787} C_VEL
LIN {X 0,Y 230.155,Z 277.317,A -85,B 0,C 180,E1 -20921.934,E2 -20921.934} C_VEL
LIN {X 0,Y 230.723,Z 278.34,A -85,B 0,C 180,E1 -20922.34,E2 -20922.34} C_VEL
LIN {X 0,Y 232.914,Z 281.973,A -85,B 0,C 180,E1 -20923.752,E2 -20923.752} C_VEL
LIN {X 0,Y 236.01,Z 287.661,A -85,B 0,C 180,E1 -20925.618,E2 -20925.618} C_VEL
LIN {X 0,Y 239.77,Z 295.216,A -85,B 0,C 180,E1 -20927.646,E2 -20927.646} C_VEL
LIN {X 0,Y 243.976,Z 305.27,A -85,B 0,C 180,E1 -20929.779,E2 -20929.779} C_VEL
LIN {X 0,Y 245.196,Z 309.013,A -85,B 0,C 180,E1 -20930.397,E2 -20930.397} C_VEL
LIN {X 0,Y 245.791,Z 319.302,A -85,B 0,C 180,E1 -20931.214,E2 -20931.214} C_VEL
LIN {X 0,Y 241.954,Z 362.101,A -85,B 0,C 180,E1 -20932.744,E2 -20932.744} C_VEL
LIN {X 0,Y 240.017,Z 374.316,A -85,B 0,C 180,E1 -20933.377,E2 -20933.377} C_VEL
LIN {X 0,Y 237.318,Z 387.208,A -85,B 0,C 180,E1 -20934.34,E2 -20934.34} C_VEL
LIN {X 0,Y 234.145,Z 398.788,A -85,B 0,C 180,E1 -20935.495,E2 -20935.495} C_VEL
LIN {X 0,Y 230.081,Z 411.3,A -85,B 0,C 180,E1 -20937.171,E2 -20937.171} C_VEL
LIN {X 0,Y 226.4,Z 421.358,A -85,B 0,C 180,E1 -20938.934,E2 -20938.934} C_VEL
LIN {X 0,Y 222.884,Z 429.717,A -85,B 0,C 180,E1 -20940.745,E2 -20940.745} C_VEL
LIN {X 0,Y 218.657,Z 438.885,A -85,B 0,C 180,E1 -20943.26,E2 -20943.26} C_VEL
LIN {X 0,Y 215.053,Z 446.388,A -85,B 0,C 180,E1 -20945.892,E2 -20945.892} C_VEL
LIN {X 0,Y 211.985,Z 452.477,A -85,B 0,C 180,E1 -20948.614,E2 -20948.614} C_VEL
LIN {X 0,Y 209.497,Z 457.349,A -85,B 0,C 180,E1 -20951.418,E2 -20951.418} C_VEL
LIN {X 0,Y 207.331,Z 461.148,A -85,B 0,C 180,E1 -20954.267,E2 -20954.267} C_VEL
LIN {X 0,Y 206.259,Z 463.152,A -85,B 0,C 180,E1 -20956.202,E2 -20956.202} C_VEL
LIN {X 0,Y 205.51,Z 464.722,A -85,B 0,C 180,E1 -20958.161,E2 -20958.161} C_VEL
LIN {X 0,Y 204.592,Z 466.644,A -85,B 0,C 180,E1 -20962.103,E2 -20962.103} C_VEL
LIN {X 0,Y 204.413,Z 467.04,A -85,B 0,C 180,E1 -20965.613,E2 -20965.613} C_VEL
LIN {X 0,Y 204.606,Z 466.566,A -85,B 0,C 180,E1 -20968.032,E2 -20968.032} C_VEL
LIN {X 0,Y 204.678,Z 465.707,A -85,B 0,C 180,E1 -20970,E2 -20970} C_VEL
LIN {X 0,Y 204.667,Z 464.423,A -85,B 0,C 180,E1 -20971.967,E2 -20971.967} C_VEL
LIN {X 0,Y 204.634,Z 461.369,A -85,B 0,C 180,E1 -20975.131,E2 -20975.131} C_VEL
LIN {X 0,Y 204.745,Z 457.65,A -85,B 0,C 180,E1 -20977.891,E2 -20977.891} C_VEL
LIN {X 0,Y 205.212,Z 452.498,A -85,B 0,C 180,E1 -20980.856,E2 -20980.856} C_VEL
LIN {X 0,Y 206.049,Z 445.931,A -85,B 0,C 180,E1 -20983.812,E2 -20983.812} C_VEL
LIN {X 0,Y 207.435,Z 437.709,A -85,B 0,C 180,E1 -20986.735,E2 -20986.735} C_VEL
LIN {X 0,Y 208.836,Z 429.276,A -85,B 0,C 180,E1 -20989.152,E2 -20989.152} C_VEL
LIN {X 0,Y 210.736,Z 418.972,A -85,B 0,C 180,E1 -20991.519,E2 -20991.519} C_VEL
LIN {X 0,Y 212.708,Z 407.353,A -85,B 0,C 180,E1 -20993.614,E2 -20993.614} C_VEL
LIN {X 0,Y 214.511,Z 396.032,A -85,B 0,C 180,E1 -20995.206,E2 -20995.206} C_VEL
LIN {X 0,Y 216.187,Z 383.319,A -85,B 0,C 180,E1 -20996.548,E2 -20996.548} C_VEL
LIN {X 0,Y 217.501,Z 370.193,A -85,B 0,C 180,E1 -20997.543,E2 -20997.543} C_VEL
LIN {X 0,Y 218.407,Z 356.415,A -85,B 0,C 180,E1 -20998.201,E2 -20998.201} C_VEL
LIN {X 0,Y 220.247,Z 311.067,A -85,B 0,C 180,E1 -20999.954,E2 -20999.954} C_VEL
LIN {X 0,Y 216.27,Z 275.893,A -85,B 0,C 180,E1 -21001.885,E2 -21001.885} C_VEL
LIN {X 0,Y 209.322,Z 255.598,A -85,B 0,C 180,E1 -21003.594,E2 -21003.594} C_VEL
LIN {X 0,Y 207.235,Z 245.849,A -85,B 0,C 180,E1 -21007.903,E2 -21007.903} C_VEL
LIN {X 0,Y 206.705,Z 243.738,A -85,B 0,C 180,E1 -21008.983,E2 -21008.983} C_VEL
LIN {X 0,Y 206.62,Z 243.751,A -85,B 0,C 180,E1 -21014.414,E2 -21014.414} C_VEL
LIN {X 0,Y 206.623,Z 243.747,A -85,B 0,C 180,E1 -21018.436,E2 -21018.436} C_VEL
LIN {X 0,Y 206.659,Z 243.742,A -85,B 0,C 180,E1 -21022.255,E2 -21022.255} C_VEL
LIN {X 0,Y 206.675,Z 243.737,A -85,B 0,C 180,E1 -21027.037,E2 -21027.037} C_VEL
LIN {X 0,Y 206.696,Z 243.733,A -85,B 0,C 180,E1 -21032.122,E2 -21032.122} C_VEL
LIN {X 0,Y 206.718,Z 243.733,A -85,B 0,C 180,E1 -21036.612,E2 -21036.612} C_VEL
LIN {X 0,Y 206.782,Z 243.719,A -85,B 0,C 180,E1 -21042.188,E2 -21042.188} C_VEL
LIN {X 0,Y 206.847,Z 243.71,A -85,B 0,C 180,E1 -21046.24,E2 -21046.24} C_VEL
LIN {X 0,Y 207.049,Z 243.692,A -85,B 0,C 180,E1 -21050.228,E2 -21050.228} C_VEL
LIN {X 0,Y 207.023,Z 243.692,A -85,B 0,C 180,E1 -21054.154,E2 -21054.154} C_VEL
LIN {X 0,Y 207.329,Z 243.639,A -85,B 0,C 180,E1 -21058.057,E2 -21058.057} C_VEL
LIN {X 0,Y 207.473,Z 243.619,A -85,B 0,C 180,E1 -21059.999,E2 -21059.999} C_VEL
LIN {X 0,Y 207.348,Z 243.643,A -85,B 0,C 180,E1 -21061.942,E2 -21061.942} C_VEL
LIN {X 0,Y 207.105,Z 243.685,A -85,B 0,C 180,E1 -21067.801,E2 -21067.801} C_VEL
LIN {X 0,Y 206.891,Z 243.708,A -85,B 0,C 180,E1 -21071.76,E2 -21071.76} C_VEL
LIN {X 0,Y 206.828,Z 243.703,A -85,B 0,C 180,E1 -21075.773,E2 -21075.773} C_VEL
LIN {X 0,Y 206.798,Z 243.696,A -85,B 0,C 180,E1 -21079.867,E2 -21079.867} C_VEL
LIN {X 0,Y 206.751,Z 243.721,A -85,B 0,C 180,E1 -21084.073,E2 -21084.073} C_VEL
LIN {X 0,Y 206.724,Z 243.736,A -85,B 0,C 180,E1 -21088.421,E2 -21088.421} C_VEL
LIN {X 0,Y 206.68,Z 243.734,A -85,B 0,C 180,E1 -21092.96,E2 -21092.96} C_VEL
LIN {X 0,Y 206.707,Z 243.715,A -85,B 0,C 180,E1 -21097.733,E2 -21097.733} C_VEL
LIN {X 0,Y 206.702,Z 243.715,A -85,B 0,C 180,E1 -21101.589,E2 -21101.589} C_VEL
LIN {X 0,Y 206.626,Z 243.741,A -85,B 0,C 180,E1 -21105.583,E2 -21105.583} C_VEL
LIN {X 0,Y 206.648,Z 243.745,A -85,B 0,C 180,E1 -21109.751,E2 -21109.751} C_VEL
LIN {X 0,Y 206.689,Z 243.728,A -85,B 0,C 180,E1 -21114.692,E2 -21114.692} C_VEL
LIN {X 0,Y 206.706,Z 243.722,A -85,B 0,C 180,E1 -21119.34,E2 -21119.34} C_VEL
LIN {X 0,Y 206.727,Z 243.735,A -85,B 0,C 180,E1 -21123.775,E2 -21123.775} C_VEL
LIN {X 0,Y 206.752,Z 243.727,A -85,B 0,C 180,E1 -21128.045,E2 -21128.045} C_VEL
LIN {X 0,Y 206.87,Z 243.708,A -85,B 0,C 180,E1 -21132.198,E2 -21132.198} C_VEL
LIN {X 0,Y 206.911,Z 243.71,A -85,B 0,C 180,E1 -21136.247,E2 -21136.247} C_VEL
LIN {X 0,Y 207.103,Z 243.678,A -85,B 0,C 180,E1 -21140.232,E2 -21140.232} C_VEL
LIN {X 0,Y 207.165,Z 243.677,A -85,B 0,C 180,E1 -21142.202,E2 -21142.202} C_VEL
LIN {X 0,Y 207.381,Z 243.649,A -85,B 0,C 180,E1 -21148.058,E2 -21148.058} C_VEL
LIN {X 0,Y 207.514,Z 243.636,A -85,B 0,C 180,E1 -21150,E2 -21150} C_VEL
LIN {X 0,Y 207.381,Z 243.65,A -85,B 0,C 180,E1 -21151.942,E2 -21151.942} C_VEL
LIN {X 0,Y 207.148,Z 243.683,A -85,B 0,C 180,E1 -21157.799,E2 -21157.799} C_VEL
LIN {X 0,Y 206.929,Z 243.711,A -85,B 0,C 180,E1 -21161.757,E2 -21161.757} C_VEL
LIN {X 0,Y 206.891,Z 243.715,A -85,B 0,C 180,E1 -21166.463,E2 -21166.463} C_VEL
LIN {X 0,Y 208.704,Z 248.431,A -85,B 0,C 180,E1 -21166.946,E2 -21166.946} C_VEL
LIN {X 0,Y 218.55,Z 271.826,A -85,B 0,C 180,E1 -21169.104,E2 -21169.104} C_VEL
LIN {X 0,Y 221.369,Z 280.025,A -85,B 0,C 180,E1 -21169.75,E2 -21169.75} C_VEL
LIN {X 0,Y 218.18,Z 345.503,A -85,B 0,C 180,E1 -21172.278,E2 -21172.278} C_VEL
LIN {X 0,Y 217.194,Z 358.879,A -85,B 0,C 180,E1 -21173.157,E2 -21173.157} C_VEL
LIN {X 0,Y 215.964,Z 371.338,A -85,B 0,C 180,E1 -21174.331,E2 -21174.331} C_VEL
LIN {X 0,Y 214.238,Z 384.537,A -85,B 0,C 180,E1 -21176.022,E2 -21176.022} C_VEL
LIN {X 0,Y 212.576,Z 395.523,A -85,B 0,C 180,E1 -21177.836,E2 -21177.836} C_VEL
LIN {X 0,Y 210.807,Z 405.919,A -85,B 0,C 180,E1 -21180.002,E2 -21180.002} C_VEL
LIN {X 0,Y 209.082,Z 415.653,A -85,B 0,C 180,E1 -21182.531,E2 -21182.531} C_VEL
LIN {X 0,Y 207.545,Z 423.766,A -85,B 0,C 180,E1 -21185.142,E2 -21185.142} C_VEL
LIN {X 0,Y 206.391,Z 430.425,A -85,B 0,C 180,E1 -21187.797,E2 -21187.797} C_VEL
LIN {X 0,Y 205.349,Z 437.025,A -85,B 0,C 180,E1 -21191.155,E2 -21191.155} C_VEL
LIN {X 0,Y 204.758,Z 441.192,A -85,B 0,C 180,E1 -21193.881,E2 -21193.881} C_VEL
LIN {X 0,Y 204.351,Z 444.352,A -85,B 0,C 180,E1 -21196.542,E2 -21196.542} C_VEL
LIN {X 0,Y 204.174,Z 446.691,A -85,B 0,C 180,E1 -21199.217,E2 -21199.217} C_VEL
LIN {X 0,Y 204.304,Z 448.404,A -85,B 0,C 180,E1 -21202.289,E2 -21202.289} C_VEL
LIN {X 0,Y 204.851,Z 449.136,A -85,B 0,C 180,E1 -21205.417,E2 -21205.417} C_VEL
LIN {X 0,Y 206.067,Z 448.64,A -85,B 0,C 180,E1 -21209.232,E2 -21209.232} C_VEL
LIN {X 0,Y 207.252,Z 447.447,A -85,B 0,C 180,E1 -21211.833,E2 -21211.833} C_VEL
LIN {X 0,Y 209.239,Z 444.873,A -85,B 0,C 180,E1 -21215.065,E2 -21215.065} C_VEL
LIN {X 0,Y 212.09,Z 440.488,A -85,B 0,C 180,E1 -21218.624,E2 -21218.624} C_VEL
LIN {X 0,Y 214.991,Z 435.676,A -85,B 0,C 180,E1 -21221.423,E2 -21221.423} C_VEL
LIN {X 0,Y 217.997,Z 430.229,A -85,B 0,C 180,E1 -21223.882,E2 -21223.882} C_VEL
LIN {X 0,Y 221.91,Z 422.269,A -85,B 0,C 180,E1 -21226.726,E2 -21226.726} C_VEL
LIN {X 0,Y 225.381,Z 414.691,A -85,B 0,C 180,E1 -21228.824,E2 -21228.824} C_VEL
LIN {X 0,Y 229.422,Z 404.777,A -85,B 0,C 180,E1 -21230.992,E2 -21230.992} C_VEL
LIN {X 0,Y 233.24,Z 393.799,A -85,B 0,C 180,E1 -21232.883,E2 -21232.883} C_VEL
LIN {X 0,Y 236.667,Z 381.831,A -85,B 0,C 180,E1 -21234.462,E2 -21234.462} C_VEL
LIN {X 0,Y 239.595,Z 369.318,A -85,B 0,C 180,E1 -21235.716,E2 -21235.716} C_VEL
LIN {X 0,Y 241.81,Z 356.056,A -85,B 0,C 180,E1 -21236.695,E2 -21236.695} C_VEL
LIN {X 0,Y 243.381,Z 343.015,A -85,B 0,C 180,E1 -21237.313,E2 -21237.313} C_VEL
LIN {X 0,Y 247.016,Z 300.696,A -85,B 0,C 180,E1 -21238.816,E2 -21238.816} C_VEL
LIN {X 0,Y 243.312,Z 292.664,A -85,B 0,C 180,E1 -21240.524,E2 -21240.524} C_VEL
LIN {X 0,Y 237.553,Z 282.087,A -85,B 0,C 180,E1 -21243.435,E2 -21243.435} C_VEL
LIN {X 0,Y 233.913,Z 276.445,A -85,B 0,C 180,E1 -21245.516,E2 -21245.516} C_VEL
LIN {X 0,Y 230.911,Z 272.676,A -85,B 0,C 180,E1 -21247.372,E2 -21247.372} C_VEL
LIN {X 0,Y 229.609,Z 270.809,A -85,B 0,C 180,E1 -21248.292,E2 -21248.292} C_VEL
LIN {X 0,Y 227.204,Z 267.397,A -85,B 0,C 180,E1 -21250.142,E2 -21250.142} C_VEL
LIN {X 0,Y 223.786,Z 263.699,A -85,B 0,C 180,E1 -21253.233,E2 -21253.233} C_VEL
LIN {X 0,Y 222.69,Z 262.356,A -85,B 0,C 180,E1 -21254.491,E2 -21254.491} C_VEL
LIN {X 0,Y 220.694,Z 260.298,A -85,B 0,C 180,E1 -21257.206,E2 -21257.206} C_VEL
LIN {X 0,Y 219.102,Z 258.542,A -85,B 0,C 180,E1 -21260.662,E2 -21260.662} C_VEL
LIN {X 0,Y 218.412,Z 258.612,A -85,B 0,C 180,E1 -21265.726,E2 -21265.726} C_VEL
LIN {X 0,Y 218.892,Z 259.491,A -85,B 0,C 180,E1 -21268.453,E2 -21268.453} C_VEL
LIN {X 0,Y 220.341,Z 261.692,A -85,B 0,C 180,E1 -21271.88,E2 -21271.88} C_VEL
LIN {X 0,Y 222.071,Z 264.683,A -85,B 0,C 180,E1 -21274.539,E2 -21274.539} C_VEL
LIN {X 0,Y 225.212,Z 269.098,A -85,B 0,C 180,E1 -21277.91,E2 -21277.91} C_VEL
LIN {X 0,Y 229.219,Z 275.529,A -85,B 0,C 180,E1 -21281.23,E2 -21281.23} C_VEL
LIN {X 0,Y 230.723,Z 278.34,A -85,B 0,C 180,E1 -21282.34,E2 -21282.34} C_VEL
LIN {X 0,Y 231.655,Z 280.895,A -85,B 0,C 180,E1 -21283.052,E2 -21283.052} C_VEL
LIN {X 0,Y 232.399,Z 286.636,A -85,B 0,C 180,E1 -21283.911,E2 -21283.911} C_VEL
LIN {X 0,Y 233.136,Z 292.506,A -85,B 0,C 180,E1 -21284.747,E2 -21284.747} C_VEL
LIN {X 0,Y 234.136,Z 295.256,A -85,B 0,C 180,E1 -21285.418,E2 -21285.418} C_VEL
LIN {X 0,Y 237.913,Z 303.712,A -85,B 0,C 180,E1 -21287.564,E2 -21287.564} C_VEL
LIN {X 0,Y 240.965,Z 312.03,A -85,B 0,C 180,E1 -21289.244,E2 -21289.244} C_VEL
LIN {X 0,Y 241.359,Z 320.657,A -85,B 0,C 180,E1 -21289.931,E2 -21289.931} C_VEL
LIN {X 0,Y 237.428,Z 362.363,A -85,B 0,C 180,E1 -21291.439,E2 -21291.439} C_VEL
LIN {X 0,Y 235.176,Z 375.701,A -85,B 0,C 180,E1 -21292.158,E2 -21292.158} C_VEL
LIN {X 0,Y 232.486,Z 387.552,A -85,B 0,C 180,E1 -21293.076,E2 -21293.076} C_VEL
LIN {X 0,Y 228.946,Z 399.628,A -85,B 0,C 180,E1 -21294.325,E2 -21294.325} C_VEL
LIN {X 0,Y 224.704,Z 411.852,A -85,B 0,C 180,E1 -21296.013,E2 -21296.013} C_VEL
LIN {X 0,Y 220.842,Z 421.72,A -85,B 0,C 180,E1 -21297.792,E2 -21297.792} C_VEL
LIN {X 0,Y 216.793,Z 430.782,A -85,B 0,C 180,E1 -21299.839,E2 -21299.839} C_VEL
LIN {X 0,Y 212.386,Z 439.711,A -85,B 0,C 180,E1 -21302.405,E2 -21302.405} C_VEL
LIN {X 0,Y 208.629,Z 446.964,A -85,B 0,C 180,E1 -21305.1,E2 -21305.1} C_VEL
LIN {X 0,Y 205.406,Z 452.848,A -85,B 0,C 180,E1 -21307.894,E2 -21307.894} C_VEL
LIN {X 0,Y 202.781,Z 457.575,A -85,B 0,C 180,E1 -21310.779,E2 -21310.779} C_VEL
LIN {X 0,Y 200.509,Z 461.237,A -85,B 0,C 180,E1 -21313.717,E2 -21313.717} C_VEL
LIN {X 0,Y 199.337,Z 463.127,A -85,B 0,C 180,E1 -21315.713,E2 -21315.713} C_VEL
LIN {X 0,Y 197.94,Z 465.686,A -85,B 0,C 180,E1 -21319.775,E2 -21319.775} C_VEL
LIN {X 0,Y 197.527,Z 466.394,A -85,B 0,C 180,E1 -21321.819,E2 -21321.819} C_VEL
LIN {X 0,Y 197.34,Z 466.623,A -85,B 0,C 180,E1 -21325.709,E2 -21325.709} C_VEL
LIN {X 0,Y 197.534,Z 466.081,A -85,B 0,C 180,E1 -21327.961,E2 -21327.961} C_VEL
LIN {X 0,Y 197.613,Z 465.163,A -85,B 0,C 180,E1 -21330,E2 -21330} C_VEL
LIN {X 0,Y 197.602,Z 463.803,A -85,B 0,C 180,E1 -21332.038,E2 -21332.038} C_VEL
LIN {X 0,Y 197.559,Z 460.898,A -85,B 0,C 180,E1 -21335.068,E2 -21335.068} C_VEL
LIN {X 0,Y 197.686,Z 456.785,A -85,B 0,C 180,E1 -21338.174,E2 -21338.174} C_VEL
LIN {X 0,Y 198.327,Z 450.439,A -85,B 0,C 180,E1 -21341.755,E2 -21341.755} C_VEL
LIN {X 0,Y 199.401,Z 443.486,A -85,B 0,C 180,E1 -21344.803,E2 -21344.803} C_VEL
LIN {X 0,Y 200.585,Z 436.344,A -85,B 0,C 180,E1 -21347.324,E2 -21347.324} C_VEL
LIN {X 0,Y 202.123,Z 427.706,A -85,B 0,C 180,E1 -21349.814,E2 -21349.814} C_VEL
LIN {X 0,Y 203.854,Z 418.339,A -85,B 0,C 180,E1 -21351.99,E2 -21351.99} C_VEL
LIN {X 0,Y 205.707,Z 407.951,A -85,B 0,C 180,E1 -21353.933,E2 -21353.933} C_VEL
LIN {X 0,Y 207.538,Z 396.841,A -85,B 0,C 180,E1 -21355.576,E2 -21355.576} C_VEL
LIN {X 0,Y 209.2,Z 384.577,A -85,B 0,C 180,E1 -21356.967,E2 -21356.967} C_VEL
LIN {X 0,Y 210.653,Z 371.205,A -85,B 0,C 180,E1 -21358.044,E2 -21358.044} C_VEL
LIN {X 0,Y 211.606,Z 358.451,A -85,B 0,C 180,E1 -21358.717,E2 -21358.717} C_VEL
LIN {X 0,Y 213.573,Z 311.542,A -85,B 0,C 180,E1 -21360.59,E2 -21360.59} C_VEL
LIN {X 0,Y 209.849,Z 277.995,A -85,B 0,C 180,E1 -21362.504,E2 -21362.504} C_VEL
LIN {X 0,Y 201.986,Z 255.166,A -85,B 0,C 180,E1 -21364.551,E2 -21364.551} C_VEL
LIN {X 0,Y 200.064,Z 246.383,A -85,B 0,C 180,E1 -21368.59,E2 -21368.59} C_VEL
LIN {X 0,Y 199.66,Z 244.615,A -85,B 0,C 180,E1 -21369.474,E2 -21369.474} C_VEL
LIN {X 0,Y 199.566,Z 244.63,A -85,B 0,C 180,E1 -21375.224,E2 -21375.224} C_VEL
LIN {X 0,Y 199.562,Z 244.628,A -85,B 0,C 180,E1 -21377.999,E2 -21377.999} C_VEL
LIN {X 0,Y 199.586,Z 244.623,A -85,B 0,C 180,E1 -21380.768,E2 -21380.768} C_VEL
LIN {X 0,Y 199.599,Z 244.62,A -85,B 0,C 180,E1 -21384.072,E2 -21384.072} C_VEL
LIN {X 0,Y 199.666,Z 244.614,A -85,B 0,C 180,E1 -21388.13,E2 -21388.13} C_VEL
LIN {X 0,Y 199.632,Z 244.613,A -85,B 0,C 180,E1 -21392.763,E2 -21392.763} C_VEL
LIN {X 0,Y 199.657,Z 244.615,A -85,B 0,C 180,E1 -21397.219,E2 -21397.219} C_VEL
LIN {X 0,Y 199.725,Z 244.598,A -85,B 0,C 180,E1 -21401.801,E2 -21401.801} C_VEL
LIN {X 0,Y 199.784,Z 244.59,A -85,B 0,C 180,E1 -21405.744,E2 -21405.744} C_VEL
LIN {X 0,Y 200.002,Z 244.571,A -85,B 0,C 180,E1 -21409.88,E2 -21409.88} C_VEL
LIN {X 0,Y 199.985,Z 244.569,A -85,B 0,C 180,E1 -21413.947,E2 -21413.947} C_VEL
LIN {X 0,Y 200.272,Z 244.517,A -85,B 0,C 180,E1 -21417.988,E2 -21417.988} C_VEL
LIN {X 0,Y 200.439,Z 244.494,A -85,B 0,C 180,E1 -21419.999,E2 -21419.999} C_VEL
LIN {X 0,Y 199.988,Z 244.566,A -85,B 0,C 180,E1 -21424.03,E2 -21424.03} C_VEL
LIN {X 0,Y 200.051,Z 244.564,A -85,B 0,C 180,E1 -21428.077,E2 -21428.077} C_VEL
LIN {X 0,Y 199.842,Z 244.587,A -85,B 0,C 180,E1 -21432.181,E2 -21432.181} C_VEL
LIN {X 0,Y 199.772,Z 244.577,A -85,B 0,C 180,E1 -21436.345,E2 -21436.345} C_VEL
LIN {X 0,Y 199.805,Z 244.563,A -85,B 0,C 180,E1 -21438.455,E2 -21438.455} C_VEL
LIN {X 0,Y 199.725,Z 244.594,A -85,B 0,C 180,E1 -21443.824,E2 -21443.824} C_VEL
LIN {X 0,Y 199.693,Z 244.611,A -85,B 0,C 180,E1 -21448.388,E2 -21448.388} C_VEL
LIN {X 0,Y 199.653,Z 244.612,A -85,B 0,C 180,E1 -21452.357,E2 -21452.357} C_VEL
LIN {X 0,Y 199.629,Z 244.599,A -85,B 0,C 180,E1 -21456.761,E2 -21456.761} C_VEL
LIN {X 0,Y 199.663,Z 244.583,A -85,B 0,C 180,E1 -21459.314,E2 -21459.314} C_VEL
LIN {X 0,Y 199.631,Z 244.6,A -85,B 0,C 180,E1 -21462.335,E2 -21462.335} C_VEL
LIN {X 0,Y 199.585,Z 244.616,A -85,B 0,C 180,E1 -21465.237,E2 -21465.237} C_VEL
LIN {X 0,Y 199.568,Z 244.626,A -85,B 0,C 180,E1 -21468.008,E2 -21468.008} C_VEL
LIN {X 0,Y 199.598,Z 244.62,A -85,B 0,C 180,E1 -21470.771,E2 -21470.771} C_VEL
LIN {X 0,Y 199.602,Z 244.606,A -85,B 0,C 180,E1 -21475.716,E2 -21475.716} C_VEL
LIN {X 0,Y 199.684,Z 244.592,A -85,B 0,C 180,E1 -21478.138,E2 -21478.138} C_VEL
LIN {X 0,Y 199.68,Z 244.609,A -85,B 0,C 180,E1 -21482.774,E2 -21482.774} C_VEL
LIN {X 0,Y 199.733,Z 244.605,A -85,B 0,C 180,E1 -21487.231,E2 -21487.231} C_VEL
LIN {X 0,Y 199.793,Z 244.587,A -85,B 0,C 180,E1 -21491.76,E2 -21491.76} C_VEL
LIN {X 0,Y 199.845,Z 244.592,A -85,B 0,C 180,E1 -21495.751,E2 -21495.751} C_VEL
LIN {X 0,Y 200.068,Z 244.555,A -85,B 0,C 180,E1 -21499.885,E2 -21499.885} C_VEL
LIN {X 0,Y 200.032,Z 244.569,A -85,B 0,C 180,E1 -21503.95,E2 -21503.95} C_VEL
LIN {X 0,Y 200.321,Z 244.529,A -85,B 0,C 180,E1 -21507.99,E2 -21507.99} C_VEL
LIN {X 0,Y 200.478,Z 244.512,A -85,B 0,C 180,E1 -21510,E2 -21510} C_VEL
LIN {X 0,Y 200.028,Z 244.568,A -85,B 0,C 180,E1 -21514.029,E2 -21514.029} C_VEL
LIN {X 0,Y 200.095,Z 244.562,A -85,B 0,C 180,E1 -21518.076,E2 -21518.076} C_VEL
LIN {X 0,Y 199.877,Z 244.59,A -85,B 0,C 180,E1 -21522.178,E2 -21522.178} C_VEL
LIN {X 0,Y 199.834,Z 244.594,A -85,B 0,C 180,E1 -21525.619,E2 -21525.619} C_VEL
LIN {X 0,Y 201.661,Z 249.314,A -85,B 0,C 180,E1 -21526.122,E2 -21526.122} C_VEL
LIN {X 0,Y 211.394,Z 272.167,A -85,B 0,C 180,E1 -21528.338,E2 -21528.338} C_VEL
LIN {X 0,Y 214.795,Z 281.746,A -85,B 0,C 180,E1 -21529.136,E2 -21529.136} C_VEL
LIN {X 0,Y 211.478,Z 345.711,A -85,B 0,C 180,E1 -21531.67,E2 -21531.67} C_VEL
LIN {X 0,Y 210.454,Z 359.076,A -85,B 0,C 180,E1 -21532.574,E2 -21532.574} C_VEL
LIN {X 0,Y 209.174,Z 371.481,A -85,B 0,C 180,E1 -21533.775,E2 -21533.775} C_VEL
LIN {X 0,Y 207.633,Z 383.064,A -85,B 0,C 180,E1 -21535.272,E2 -21535.272} C_VEL
LIN {X 0,Y 205.708,Z 395.458,A -85,B 0,C 180,E1 -21537.343,E2 -21537.343} C_VEL
LIN {X 0,Y 203.974,Z 405.57,A -85,B 0,C 180,E1 -21539.491,E2 -21539.491} C_VEL
LIN {X 0,Y 202.206,Z 415.071,A -85,B 0,C 180,E1 -21542.004,E2 -21542.004} C_VEL
LIN {X 0,Y 200.458,Z 424.241,A -85,B 0,C 180,E1 -21545.032,E2 -21545.032} C_VEL
LIN {X 0,Y 199.006,Z 432.15,A -85,B 0,C 180,E1 -21548.401,E2 -21548.401} C_VEL
LIN {X 0,Y 198.104,Z 438.411,A -85,B 0,C 180,E1 -21551.842,E2 -21551.842} C_VEL
LIN {X 0,Y 197.406,Z 443.204,A -85,B 0,C 180,E1 -21555.394,E2 -21555.394} C_VEL
LIN {X 0,Y 197.1,Z 446.211,A -85,B 0,C 180,E1 -21558.479,E2 -21558.479} C_VEL
LIN {X 0,Y 197.147,Z 448.267,A -85,B 0,C 180,E1 -21561.645,E2 -21561.645} C_VEL
LIN {X 0,Y 197.736,Z 449.409,A -85,B 0,C 180,E1 -21565.343,E2 -21565.343} C_VEL
LIN {X 0,Y 198.533,Z 449.415,A -85,B 0,C 180,E1 -21568.157,E2 -21568.157} C_VEL
LIN {X 0,Y 199.931,Z 448.407,A -85,B 0,C 180,E1 -21571.487,E2 -21571.487} C_VEL
LIN {X 0,Y 202.271,Z 445.793,A -85,B 0,C 180,E1 -21575.359,E2 -21575.359} C_VEL
LIN {X 0,Y 205.29,Z 441.607,A -85,B 0,C 180,E1 -21579.102,E2 -21579.102} C_VEL
LIN {X 0,Y 208.765,Z 436.306,A -85,B 0,C 180,E1 -21582.364,E2 -21582.364} C_VEL
LIN {X 0,Y 212.26,Z 430.369,A -85,B 0,C 180,E1 -21585.132,E2 -21585.132} C_VEL
LIN {X 0,Y 215.837,Z 423.589,A -85,B 0,C 180,E1 -21587.619,E2 -21587.619} C_VEL
LIN {X 0,Y 219.546,Z 416.016,A -85,B 0,C 180,E1 -21589.808,E2 -21589.808} C_VEL
LIN {X 0,Y 223.486,Z 407.043,A -85,B 0,C 180,E1 -21591.865,E2 -21591.865} C_VEL
LIN {X 0,Y 227.721,Z 395.757,A -85,B 0,C 180,E1 -21593.91,E2 -21593.91} C_VEL
LIN {X 0,Y 230.995,Z 385.5,A -85,B 0,C 180,E1 -21595.363,E2 -21595.363} C_VEL
LIN {X 0,Y 234.149,Z 373.531,A -85,B 0,C 180,E1 -21596.667,E2 -21596.667} C_VEL
LIN {X 0,Y 236.498,Z 361.628,A -85,B 0,C 180,E1 -21597.659,E2 -21597.659} C_VEL
LIN {X 0,Y 238.314,Z 349.163,A -85,B 0,C 180,E1 -21598.391,E2 -21598.391} C_VEL
LIN {X 0,Y 242.555,Z 303.771,A -85,B 0,C 180,E1 -21600.031,E2 -21600.031} C_VEL
LIN {X 0,Y 239.312,Z 296.581,A -85,B 0,C 180,E1 -21601.683,E2 -21601.683} C_VEL
LIN {X 0,Y 234.607,Z 287.598,A -85,B 0,C 180,E1 -21604.266,E2 -21604.266} C_VEL
LIN {X 0,Y 231.296,Z 282.512,A -85,B 0,C 180,E1 -21606.237,E2 -21606.237} C_VEL
LIN {X 0,Y 228.394,Z 278.405,A -85,B 0,C 180,E1 -21608.215,E2 -21608.215} C_VEL
LIN {X 0,Y 224.863,Z 273.382,A -85,B 0,C 180,E1 -21611.06,E2 -21611.06} C_VEL
LIN {X 0,Y 222.251,Z 270.558,A -85,B 0,C 180,E1 -21613.547,E2 -21613.547} C_VEL
LIN {X 0,Y 221.148,Z 269.076,A -85,B 0,C 180,E1 -21614.906,E2 -21614.906} C_VEL
LIN {X 0,Y 219.303,Z 267.139,A -85,B 0,C 180,E1 -21617.548,E2 -21617.548} C_VEL
LIN {X 0,Y 217.886,Z 265.53,A -85,B 0,C 180,E1 -21620.782,E2 -21620.782} C_VEL
LIN {X 0,Y 217.28,Z 265.658,A -85,B 0,C 180,E1 -21626.036,E2 -21626.036} C_VEL
LIN {X 0,Y 217.86,Z 266.787,A -85,B 0,C 180,E1 -21628.94,E2 -21628.94} C_VEL
LIN {X 0,Y 219.032,Z 268.645,A -85,B 0,C 180,E1 -21631.681,E2 -21631.681} C_VEL
LIN {X 0,Y 223.14,Z 275.198,A -85,B 0,C 180,E1 -21637.125,E2 -21637.125} C_VEL
LIN {X 0,Y 226.975,Z 281.739,A -85,B 0,C 180,E1 -21640.56,E2 -21640.56} C_VEL
LIN {X 0,Y 230.366,Z 287.981,A -85,B 0,C 180,E1 -21643.053,E2 -21643.053} C_VEL
LIN {X 0,Y 233.338,Z 293.673,A -85,B 0,C 180,E1 -21644.935,E2 -21644.935} C_VEL
LIN {X 0,Y 234.136,Z 295.256,A -85,B 0,C 180,E1 -21645.418,E2 -21645.418} C_VEL
LIN {X 0,Y 234.975,Z 297.493,A -85,B 0,C 180,E1 -21645.955,E2 -21645.955} C_VEL
LIN {X 0,Y 235.499,Z 301.568,A -85,B 0,C 180,E1 -21646.48,E2 -21646.48} C_VEL
LIN {X 0,Y 235.842,Z 310.594,A -85,B 0,C 180,E1 -21647.284,E2 -21647.284} C_VEL
LIN {X 0,Y 236.525,Z 314.042,A -85,B 0,C 180,E1 -21647.792,E2 -21647.792} C_VEL
LIN {X 0,Y 236.952,Z 315.551,A -85,B 0,C 180,E1 -21648.058,E2 -21648.058} C_VEL
LIN {X 0,Y 237.18,Z 321.654,A -85,B 0,C 180,E1 -21648.576,E2 -21648.576} C_VEL
LIN {X 0,Y 233.198,Z 361.55,A -85,B 0,C 180,E1 -21650.038,E2 -21650.038} C_VEL
LIN {X 0,Y 230.962,Z 374.395,A -85,B 0,C 180,E1 -21650.71,E2 -21650.71} C_VEL
LIN {X 0,Y 228.051,Z 386.982,A -85,B 0,C 180,E1 -21651.674,E2 -21651.674} C_VEL
LIN {X 0,Y 224.353,Z 399.117,A -85,B 0,C 180,E1 -21652.918,E2 -21652.918} C_VEL
LIN {X 0,Y 220.425,Z 410.113,A -85,B 0,C 180,E1 -21654.422,E2 -21654.422} C_VEL
LIN {X 0,Y 215.81,Z 421.22,A -85,B 0,C 180,E1 -21656.389,E2 -21656.389} C_VEL
LIN {X 0,Y 210.759,Z 431.854,A -85,B 0,C 180,E1 -21658.881,E2 -21658.881} C_VEL
LIN {X 0,Y 206.172,Z 440.524,A -85,B 0,C 180,E1 -21661.498,E2 -21661.498} C_VEL
LIN {X 0,Y 201.62,Z 448.556,A -85,B 0,C 180,E1 -21664.725,E2 -21664.725} C_VEL
LIN {X 0,Y 197.86,Z 454.872,A -85,B 0,C 180,E1 -21668.104,E2 -21668.104} C_VEL
LIN {X 0,Y 195.238,Z 459.049,A -85,B 0,C 180,E1 -21671.099,E2 -21671.099} C_VEL
LIN {X 0,Y 193.677,Z 461.281,A -85,B 0,C 180,E1 -21673.126,E2 -21673.126} C_VEL
LIN {X 0,Y 192.432,Z 463.08,A -85,B 0,C 180,E1 -21675.189,E2 -21675.189} C_VEL
LIN {X 0,Y 190.941,Z 465.511,A -85,B 0,C 180,E1 -21679.396,E2 -21679.396} C_VEL
LIN {X 0,Y 190.484,Z 466.126,A -85,B 0,C 180,E1 -21681.514,E2 -21681.514} C_VEL
LIN {X 0,Y 190.263,Z 466.158,A -85,B 0,C 180,E1 -21685.764,E2 -21685.764} C_VEL
LIN {X 0,Y 190.462,Z 465.597,A -85,B 0,C 180,E1 -21687.885,E2 -21687.885} C_VEL
LIN {X 0,Y 190.549,Z 464.611,A -85,B 0,C 180,E1 -21690,E2 -21690} C_VEL
LIN {X 0,Y 190.539,Z 463.136,A -85,B 0,C 180,E1 -21692.113,E2 -21692.113} C_VEL
LIN {X 0,Y 190.498,Z 460.347,A -85,B 0,C 180,E1 -21695.051,E2 -21695.051} C_VEL
LIN {X 0,Y 190.655,Z 455.843,A -85,B 0,C 180,E1 -21698.478,E2 -21698.478} C_VEL
LIN {X 0,Y 191.328,Z 449.333,A -85,B 0,C 180,E1 -21702.192,E2 -21702.192} C_VEL
LIN {X 0,Y 192.488,Z 442.173,A -85,B 0,C 180,E1 -21705.348,E2 -21705.348} C_VEL
LIN {X 0,Y 194.081,Z 433.159,A -85,B 0,C 180,E1 -21708.47,E2 -21708.47} C_VEL
LIN {X 0,Y 195.859,Z 423.926,A -85,B 0,C 180,E1 -21711.026,E2 -21711.026} C_VEL
LIN {X 0,Y 197.725,Z 413.683,A -85,B 0,C 180,E1 -21713.29,E2 -21713.29} C_VEL
LIN {X 0,Y 199.69,Z 402.403,A -85,B 0,C 180,E1 -21715.257,E2 -21715.257} C_VEL
LIN {X 0,Y 201.745,Z 389.929,A -85,B 0,C 180,E1 -21716.924,E2 -21716.924} C_VEL
LIN {X 0,Y 203.375,Z 376.569,A -85,B 0,C 180,E1 -21718.225,E2 -21718.225} C_VEL
LIN {X 0,Y 204.573,Z 363.532,A -85,B 0,C 180,E1 -21719.096,E2 -21719.096} C_VEL
LIN {X 0,Y 206.953,Z 312.576,A -85,B 0,C 180,E1 -21721.23,E2 -21721.23} C_VEL
LIN {X 0,Y 203.486,Z 280.188,A -85,B 0,C 180,E1 -21723.117,E2 -21723.117} C_VEL
LIN {X 0,Y 195.384,Z 257.155,A -85,B 0,C 180,E1 -21725.245,E2 -21725.245} C_VEL
LIN {X 0,Y 194.681,Z 254.894,A -85,B 0,C 180,E1 -21725.481,E2 -21725.481} C_VEL
LIN {X 0,Y 192.884,Z 246.906,A -85,B 0,C 180,E1 -21729.32,E2 -21729.32} C_VEL
LIN {X 0,Y 192.59,Z 245.497,A -85,B 0,C 180,E1 -21730.113,E2 -21730.113} C_VEL
LIN {X 0,Y 192.479,Z 245.513,A -85,B 0,C 180,E1 -21733.921,E2 -21733.921} C_VEL
LIN {X 0,Y 192.495,Z 245.507,A -85,B 0,C 180,E1 -21738.914,E2 -21738.914} C_VEL
LIN {X 0,Y 192.57,Z 245.499,A -85,B 0,C 180,E1 -21743.4,E2 -21743.4} C_VEL
LIN {X 0,Y 192.589,Z 245.491,A -85,B 0,C 180,E1 -21747.058,E2 -21747.058} C_VEL
LIN {X 0,Y 192.62,Z 245.488,A -85,B 0,C 180,E1 -21751.684,E2 -21751.684} C_VEL
LIN {X 0,Y 192.652,Z 245.485,A -85,B 0,C 180,E1 -21756.341,E2 -21756.341} C_VEL
LIN {X 0,Y 192.675,Z 245.478,A -85,B 0,C 180,E1 -21761.49,E2 -21761.49} C_VEL
LIN {X 0,Y 192.709,Z 245.465,A -85,B 0,C 180,E1 -21765.209,E2 -21765.209} C_VEL
LIN {X 0,Y 192.925,Z 245.453,A -85,B 0,C 180,E1 -21769.565,E2 -21769.565} C_VEL
LIN {X 0,Y 192.948,Z 245.445,A -85,B 0,C 180,E1 -21773.726,E2 -21773.726} C_VEL
LIN {X 0,Y 193.216,Z 245.395,A -85,B 0,C 180,E1 -21777.915,E2 -21777.915} C_VEL
LIN {X 0,Y 193.404,Z 245.369,A -85,B 0,C 180,E1 -21779.999,E2 -21779.999} C_VEL
LIN {X 0,Y 192.934,Z 245.444,A -85,B 0,C 180,E1 -21784.177,E2 -21784.177} C_VEL
LIN {X 0,Y 193.002,Z 245.443,A -85,B 0,C 180,E1 -21788.375,E2 -21788.375} C_VEL
LIN {X 0,Y 192.77,Z 245.465,A -85,B 0,C 180,E1 -21792.635,E2 -21792.635} C_VEL
LIN {X 0,Y 192.742,Z 245.446,A -85,B 0,C 180,E1 -21796.959,E2 -21796.959} C_VEL
LIN {X 0,Y 192.653,Z 245.466,A -85,B 0,C 180,E1 -21801.395,E2 -21801.395} C_VEL
LIN {X 0,Y 192.651,Z 245.477,A -85,B 0,C 180,E1 -21804.23,E2 -21804.23} C_VEL
LIN {X 0,Y 192.63,Z 245.489,A -85,B 0,C 180,E1 -21808.893,E2 -21808.893} C_VEL
LIN {X 0,Y 192.579,Z 245.49,A -85,B 0,C 180,E1 -21813.189,E2 -21813.189} C_VEL
LIN {X 0,Y 192.582,Z 245.466,A -85,B 0,C 180,E1 -21818.344,E2 -21818.344} C_VEL
LIN {X 0,Y 192.549,Z 245.485,A -85,B 0,C 180,E1 -21823.121,E2 -21823.121} C_VEL
LIN {X 0,Y 192.505,Z 245.503,A -85,B 0,C 180,E1 -21826.899,E2 -21826.899} C_VEL
LIN {X 0,Y 192.54,Z 245.501,A -85,B 0,C 180,E1 -21831.651,E2 -21831.651} C_VEL
LIN {X 0,Y 192.588,Z 245.474,A -85,B 0,C 180,E1 -21836.817,E2 -21836.817} C_VEL
LIN {X 0,Y 192.658,Z 245.481,A -85,B 0,C 180,E1 -21841.694,E2 -21841.694} C_VEL
LIN {X 0,Y 192.7,Z 245.48,A -85,B 0,C 180,E1 -21846.351,E2 -21846.351} C_VEL
LIN {X 0,Y 192.728,Z 245.465,A -85,B 0,C 180,E1 -21851.46,E2 -21851.46} C_VEL
LIN {X 0,Y 192.769,Z 245.472,A -85,B 0,C 180,E1 -21855.216,E2 -21855.216} C_VEL
LIN {X 0,Y 192.979,Z 245.44,A -85,B 0,C 180,E1 -21859.51,E2 -21859.51} C_VEL
LIN {X 0,Y 193.06,Z 245.432,A -85,B 0,C 180,E1 -21861.628,E2 -21861.628} C_VEL
LIN {X 0,Y 193.262,Z 245.408,A -85,B 0,C 180,E1 -21867.916,E2 -21867.916} C_VEL
LIN {X 0,Y 193.442,Z 245.389,A -85,B 0,C 180,E1 -21870,E2 -21870} C_VEL
LIN {X 0,Y 192.975,Z 245.446,A -85,B 0,C 180,E1 -21874.177,E2 -21874.177} C_VEL
LIN {X 0,Y 193.045,Z 245.441,A -85,B 0,C 180,E1 -21878.373,E2 -21878.373} C_VEL
LIN {X 0,Y 192.804,Z 245.471,A -85,B 0,C 180,E1 -21882.632,E2 -21882.632} C_VEL
LIN {X 0,Y 192.783,Z 245.473,A -85,B 0,C 180,E1 -21884.716,E2 -21884.716} C_VEL
LIN {X 0,Y 193.903,Z 248.49,A -85,B 0,C 180,E1 -21885.065,E2 -21885.065} C_VEL
LIN {X 0,Y 203.016,Z 269.741,A -85,B 0,C 180,E1 -21887.27,E2 -21887.27} C_VEL
LIN {X 0,Y 207.36,Z 280.906,A -85,B 0,C 180,E1 -21888.292,E2 -21888.292} C_VEL
LIN {X 0,Y 208.072,Z 282.939,A -85,B 0,C 180,E1 -21888.464,E2 -21888.464} C_VEL
LIN {X 0,Y 204.733,Z 346.499,A -85,B 0,C 180,E1 -21891.092,E2 -21891.092} C_VEL
LIN {X 0,Y 203.691,Z 359.532,A -85,B 0,C 180,E1 -21892.008,E2 -21892.008} C_VEL
LIN {X 0,Y 202.339,Z 372.101,A -85,B 0,C 180,E1 -21893.269,E2 -21893.269} C_VEL
LIN {X 0,Y 200.563,Z 384.832,A -85,B 0,C 180,E1 -21895.001,E2 -21895.001} C_VEL
LIN {X 0,Y 198.613,Z 396.73,A -85,B 0,C 180,E1 -21897.1,E2 -21897.1} C_VEL
LIN {X 0,Y 196.739,Z 407.033,A -85,B 0,C 180,E1 -21899.419,E2 -21899.419} C_VEL
LIN {X 0,Y 194.887,Z 416.977,A -85,B 0,C 180,E1 -21902.215,E2 -21902.215} C_VEL
LIN {X 0,Y 193.29,Z 425.098,A -85,B 0,C 180,E1 -21905.078,E2 -21905.078} C_VEL
LIN {X 0,Y 191.832,Z 432.809,A -85,B 0,C 180,E1 -21908.517,E2 -21908.517} C_VEL
LIN {X 0,Y 191.068,Z 438.001,A -85,B 0,C 180,E1 -21911.454,E2 -21911.454} C_VEL
LIN {X 0,Y 190.436,Z 442.276,A -85,B 0,C 180,E1 -21914.517,E2 -21914.517} C_VEL
LIN {X 0,Y 190.009,Z 446.124,A -85,B 0,C 180,E1 -21918.259,E2 -21918.259} C_VEL
LIN {X 0,Y 190.01,Z 448.048,A -85,B 0,C 180,E1 -21921.04,E2 -21921.04} C_VEL
LIN {X 0,Y 190.388,Z 449.426,A -85,B 0,C 180,E1 -21924.294,E2 -21924.294} C_VEL
LIN {X 0,Y 191.255,Z 449.858,A -85,B 0,C 180,E1 -21927.681,E2 -21927.681} C_VEL
LIN {X 0,Y 192.932,Z 449.03,A -85,B 0,C 180,E1 -21931.736,E2 -21931.736} C_VEL
LIN {X 0,Y 194.544,Z 447.501,A -85,B 0,C 180,E1 -21934.56,E2 -21934.56} C_VEL
LIN {X 0,Y 197.081,Z 444.582,A -85,B 0,C 180,E1 -21937.982,E2 -21937.982} C_VEL
LIN {X 0,Y 200.577,Z 439.925,A -85,B 0,C 180,E1 -21941.619,E2 -21941.619} C_VEL
LIN {X 0,Y 204.124,Z 434.674,A -85,B 0,C 180,E1 -21944.566,E2 -21944.566} C_VEL
LIN {X 0,Y 208.549,Z 427.228,A -85,B 0,C 180,E1 -21947.736,E2 -21947.736} C_VEL
LIN {X 0,Y 212.199,Z 420.437,A -85,B 0,C 180,E1 -21949.987,E2 -21949.987} C_VEL
LIN {X 0,Y 216.581,Z 411.551,A -85,B 0,C 180,E1 -21952.308,E2 -21952.308} C_VEL
LIN {X 0,Y 221.311,Z 400.451,A -85,B 0,C 180,E1 -21954.534,E2 -21954.534} C_VEL
LIN {X 0,Y 225.137,Z 389.702,A -85,B 0,C 180,E1 -21956.22,E2 -21956.22} C_VEL
LIN {X 0,Y 228.787,Z 377.267,A -85,B 0,C 180,E1 -21957.69,E2 -21957.69} C_VEL
LIN {X 0,Y 231.746,Z 363.974,A -85,B 0,C 180,E1 -21958.887,E2 -21958.887} C_VEL
LIN {X 0,Y 233.876,Z 350.663,A -85,B 0,C 180,E1 -21959.712,E2 -21959.712} C_VEL
LIN {X 0,Y 238.152,Z 308.543,A -85,B 0,C 180,E1 -21961.254,E2 -21961.254} C_VEL
LIN {X 0,Y 238.26,Z 306.603,A -85,B 0,C 180,E1 -21961.353,E2 -21961.353} C_VEL
LIN {X 0,Y 234.574,Z 298.902,A -85,B 0,C 180,E1 -21963.354,E2 -21963.354} C_VEL
LIN {X 0,Y 231.589,Z 292.948,A -85,B 0,C 180,E1 -21965.181,E2 -21965.181} C_VEL
LIN {X 0,Y 228.809,Z 288.562,A -85,B 0,C 180,E1 -21966.965,E2 -21966.965} C_VEL
LIN {X 0,Y 226.034,Z 284.366,A -85,B 0,C 180,E1 -21968.986,E2 -21968.986} C_VEL
LIN {X 0,Y 222.96,Z 279.931,A -85,B 0,C 180,E1 -21971.637,E2 -21971.637} C_VEL
LIN {X 0,Y 220.602,Z 277.178,A -85,B 0,C 180,E1 -21974.049,E2 -21974.049} C_VEL
LIN {X 0,Y 219.583,Z 275.778,A -85,B 0,C 180,E1 -21975.371,E2 -21975.371} C_VEL
LIN {X 0,Y 217.928,Z 273.999,A -85,B 0,C 180,E1 -21977.893,E2 -21977.893} C_VEL
LIN {X 0,Y 216.674,Z 272.507,A -85,B 0,C 180,E1 -21980.904,E2 -21980.904} C_VEL
LIN {X 0,Y 216.092,Z 272.624,A -85,B 0,C 180,E1 -21985.776,E2 -21985.776} C_VEL
LIN {X 0,Y 216.569,Z 273.655,A -85,B 0,C 180,E1 -21988.578,E2 -21988.578} C_VEL
LIN {X 0,Y 217.672,Z 275.498,A -85,B 0,C 180,E1 -21991.365,E2 -21991.365} C_VEL
LIN {X 0,Y 221.328,Z 281.74,A -85,B 0,C 180,E1 -21996.569,E2 -21996.569} C_VEL
LIN {X 0,Y 224.764,Z 287.973,A -85,B 0,C 180,E1 -21999.882,E2 -21999.882} C_VEL
LIN {X 0,Y 227.896,Z 294.028,A -85,B 0,C 180,E1 -22002.338,E2 -22002.338} C_VEL
LIN {X 0,Y 230.596,Z 299.47,A -85,B 0,C 180,E1 -22004.172,E2 -22004.172} C_VEL
LIN {X 0,Y 234.272,Z 307.964,A -85,B 0,C 180,E1 -22006.481,E2 -22006.481} C_VEL
LIN {X 0,Y 236.525,Z 314.042,A -85,B 0,C 180,E1 -22007.792,E2 -22007.792} C_VEL
LIN {X 0,Y 236.813,Z 316.229,A -85,B 0,C 180,E1 -22008.056,E2 -22008.056} C_VEL
LIN {X 0,Y 236.322,Z 320.01,A -85,B 0,C 180,E1 -22008.147,E2 -22008.147} C_VEL
LIN {X 0,Y 235.212,Z 323.803,A -85,B 0,C 180,E1 -22008.011,E2 -22008.011} C_VEL
LIN {X 0,Y 232.853,Z 330.594,A -85,B 0,C 180,E1 -22007.623,E2 -22007.623} C_VEL
LIN {X 0,Y 231.962,Z 334.832,A -85,B 0,C 180,E1 -22007.596,E2 -22007.596} C_VEL
LIN {X 0,Y 229.029,Z 362.212,A -85,B 0,C 180,E1 -22008.627,E2 -22008.627} C_VEL
LIN {X 0,Y 226.899,Z 373.691,A -85,B 0,C 180,E1 -22009.227,E2 -22009.227} C_VEL
LIN {X 0,Y 223.783,Z 386.63,A -85,B 0,C 180,E1 -22010.222,E2 -22010.222} C_VEL
LIN {X 0,Y 219.906,Z 398.692,A -85,B 0,C 180,E1 -22011.455,E2 -22011.455} C_VEL
LIN {X 0,Y 215.817,Z 409.632,A -85,B 0,C 180,E1 -22012.959,E2 -22012.959} C_VEL
LIN {X 0,Y 211.433,Z 419.765,A -85,B 0,C 180,E1 -22014.726,E2 -22014.726} C_VEL
LIN {X 0,Y 206.495,Z 429.818,A -85,B 0,C 180,E1 -22017.01,E2 -22017.01} C_VEL
LIN {X 0,Y 201.591,Z 438.728,A -85,B 0,C 180,E1 -22019.638,E2 -22019.638} C_VEL
LIN {X 0,Y 197.226,Z 445.989,A -85,B 0,C 180,E1 -22022.407,E2 -22022.407} C_VEL
LIN {X 0,Y 192.936,Z 452.748,A -85,B 0,C 180,E1 -22025.805,E2 -22025.805} C_VEL
LIN {X 0,Y 189.4,Z 457.968,A -85,B 0,C 180,E1 -22029.361,E2 -22029.361} C_VEL
LIN {X 0,Y 186.874,Z 461.331,A -85,B 0,C 180,E1 -22032.492,E2 -22032.492} C_VEL
LIN {X 0,Y 185.545,Z 463.047,A -85,B 0,C 180,E1 -22034.626,E2 -22034.626} C_VEL
LIN {X 0,Y 184.627,Z 464.378,A -85,B 0,C 180,E1 -22036.799,E2 -22036.799} C_VEL
LIN {X 0,Y 183.929,Z 465.3,A -85,B 0,C 180,E1 -22038.987,E2 -22038.987} C_VEL
LIN {X 0,Y 183.203,Z 465.96,A -85,B 0,C 180,E1 -22043.392,E2 -22043.392} C_VEL
LIN {X 0,Y 183.39,Z 465.091,A -85,B 0,C 180,E1 -22047.804,E2 -22047.804} C_VEL
LIN {X 0,Y 183.487,Z 463.996,A -85,B 0,C 180,E1 -22050,E2 -22050} C_VEL
LIN {X 0,Y 183.475,Z 462.458,A -85,B 0,C 180,E1 -22052.195,E2 -22052.195} C_VEL
LIN {X 0,Y 183.419,Z 459.86,A -85,B 0,C 180,E1 -22054.967,E2 -22054.967} C_VEL
LIN {X 0,Y 183.616,Z 454.896,A -85,B 0,C 180,E1 -22058.806,E2 -22058.806} C_VEL
LIN {X 0,Y 184.22,Z 449.263,A -85,B 0,C 180,E1 -22062.111,E2 -22062.111} C_VEL
LIN {X 0,Y 185.359,Z 442.179,A -85,B 0,C 180,E1 -22065.389,E2 -22065.389} C_VEL
LIN {X 0,Y 186.977,Z 433.238,A -85,B 0,C 180,E1 -22068.63,E2 -22068.63} C_VEL
LIN {X 0,Y 188.879,Z 423.689,A -85,B 0,C 180,E1 -22071.383,E2 -22071.383} C_VEL
LIN {X 0,Y 190.699,Z 413.986,A -85,B 0,C 180,E1 -22073.624,E2 -22073.624} C_VEL
LIN {X 0,Y 192.699,Z 402.837,A -85,B 0,C 180,E1 -22075.661,E2 -22075.661} C_VEL
LIN {X 0,Y 194.799,Z 390.578,A -85,B 0,C 180,E1 -22077.383,E2 -22077.383} C_VEL
LIN {X 0,Y 196.452,Z 377.621,A -85,B 0,C 180,E1 -22078.729,E2 -22078.729} C_VEL
LIN {X 0,Y 197.755,Z 364.176,A -85,B 0,C 180,E1 -22079.687,E2 -22079.687} C_VEL
LIN {X 0,Y 200.296,Z 313.287,A -85,B 0,C 180,E1 -22081.901,E2 -22081.901} C_VEL
LIN {X 0,Y 196.934,Z 281.94,A -85,B 0,C 180,E1 -22083.814,E2 -22083.814} C_VEL
LIN {X 0,Y 189.22,Z 259.794,A -85,B 0,C 180,E1 -22085.942,E2 -22085.942} C_VEL
LIN {X 0,Y 187.372,Z 254.506,A -85,B 0,C 180,E1 -22086.524,E2 -22086.524} C_VEL
LIN {X 0,Y 185.522,Z 246.375,A -85,B 0,C 180,E1 -22090.742,E2 -22090.742} C_VEL
LIN {X 0,Y 185.446,Z 246.389,A -85,B 0,C 180,E1 -22096.052,E2 -22096.052} C_VEL
LIN {X 0,Y 185.446,Z 246.387,A -85,B 0,C 180,E1 -22099.889,E2 -22099.889} C_VEL
LIN {X 0,Y 185.488,Z 246.379,A -85,B 0,C 180,E1 -22102.71,E2 -22102.71} C_VEL
LIN {X 0,Y 185.516,Z 246.377,A -85,B 0,C 180,E1 -22107.969,E2 -22107.969} C_VEL
LIN {X 0,Y 185.536,Z 246.373,A -85,B 0,C 180,E1 -22110.59,E2 -22110.59} C_VEL
LIN {X 0,Y 185.564,Z 246.365,A -85,B 0,C 180,E1 -22115.378,E2 -22115.378} C_VEL
LIN {X 0,Y 185.606,Z 246.36,A -85,B 0,C 180,E1 -22121.177,E2 -22121.177} C_VEL
LIN {X 0,Y 185.64,Z 246.342,A -85,B 0,C 180,E1 -22124.632,E2 -22124.632} C_VEL
LIN {X 0,Y 185.868,Z 246.333,A -85,B 0,C 180,E1 -22129.418,E2 -22129.418} C_VEL
LIN {X 0,Y 185.912,Z 246.322,A -85,B 0,C 180,E1 -22133.487,E2 -22133.487} C_VEL
LIN {X 0,Y 186.162,Z 246.273,A -85,B 0,C 180,E1 -22137.836,E2 -22137.836} C_VEL
LIN {X 0,Y 186.369,Z 246.244,A -85,B 0,C 180,E1 -22139.999,E2 -22139.999} C_VEL
LIN {X 0,Y 185.881,Z 246.323,A -85,B 0,C 180,E1 -22144.336,E2 -22144.336} C_VEL
LIN {X 0,Y 185.952,Z 246.323,A -85,B 0,C 180,E1 -22148.694,E2 -22148.694} C_VEL
LIN {X 0,Y 185.698,Z 246.342,A -85,B 0,C 180,E1 -22153.124,E2 -22153.124} C_VEL
LIN {X 0,Y 185.691,Z 246.317,A -85,B 0,C 180,E1 -22158.9,E2 -22158.9} C_VEL
LIN {X 0,Y 185.588,Z 246.359,A -85,B 0,C 180,E1 -22164.617,E2 -22164.617} C_VEL
LIN {X 0,Y 185.561,Z 246.369,A -85,B 0,C 180,E1 -22169.495,E2 -22169.495} C_VEL
LIN {X 0,Y 185.495,Z 246.367,A -85,B 0,C 180,E1 -22174.632,E2 -22174.632} C_VEL
LIN {X 0,Y 185.529,Z 246.352,A -85,B 0,C 180,E1 -22177.307,E2 -22177.307} C_VEL
LIN {X 0,Y 185.517,Z 246.346,A -85,B 0,C 180,E1 -22180.749,E2 -22180.749} C_VEL
LIN {X 0,Y 185.503,Z 246.365,A -85,B 0,C 180,E1 -22183.966,E2 -22183.966} C_VEL
LIN {X 0,Y 185.46,Z 246.382,A -85,B 0,C 180,E1 -22189.278,E2 -22189.278} C_VEL
LIN {X 0,Y 185.495,Z 246.373,A -85,B 0,C 180,E1 -22192.715,E2 -22192.715} C_VEL
LIN {X 0,Y 185.535,Z 246.351,A -85,B 0,C 180,E1 -22197.977,E2 -22197.977} C_VEL
LIN {X 0,Y 185.575,Z 246.36,A -85,B 0,C 180,E1 -22200.579,E2 -22200.579} C_VEL
LIN {X 0,Y 185.582,Z 246.369,A -85,B 0,C 180,E1 -22205.385,E2 -22205.385} C_VEL
LIN {X 0,Y 185.671,Z 246.343,A -85,B 0,C 180,E1 -22211.135,E2 -22211.135} C_VEL
LIN {X 0,Y 185.721,Z 246.348,A -85,B 0,C 180,E1 -22214.641,E2 -22214.641} C_VEL
LIN {X 0,Y 185.922,Z 246.32,A -85,B 0,C 180,E1 -22219.36,E2 -22219.36} C_VEL
LIN {X 0,Y 185.959,Z 246.323,A -85,B 0,C 180,E1 -22223.491,E2 -22223.491} C_VEL
LIN {X 0,Y 186.207,Z 246.287,A -85,B 0,C 180,E1 -22227.837,E2 -22227.837} C_VEL
LIN {X 0,Y 186.406,Z 246.266,A -85,B 0,C 180,E1 -22230,E2 -22230} C_VEL
LIN {X 0,Y 185.921,Z 246.325,A -85,B 0,C 180,E1 -22234.336,E2 -22234.336} C_VEL
LIN {X 0,Y 185.991,Z 246.321,A -85,B 0,C 180,E1 -22238.693,E2 -22238.693} C_VEL
LIN {X 0,Y 185.767,Z 246.375,A -85,B 0,C 180,E1 -22243.815,E2 -22243.815} C_VEL
LIN {X 0,Y 186.797,Z 249.277,A -85,B 0,C 180,E1 -22244.118,E2 -22244.118} C_VEL
LIN {X 0,Y 195.231,Z 268.388,A -85,B 0,C 180,E1 -22246.232,E2 -22246.232} C_VEL
LIN {X 0,Y 201.03,Z 283.211,A -85,B 0,C 180,E1 -22247.675,E2 -22247.675} C_VEL
LIN {X 0,Y 201.471,Z 285.39,A -85,B 0,C 180,E1 -22247.831,E2 -22247.831} C_VEL
LIN {X 0,Y 197.99,Z 346.942,A -85,B 0,C 180,E1 -22250.449,E2 -22250.449} C_VEL
LIN {X 0,Y 196.956,Z 359.737,A -85,B 0,C 180,E1 -22251.38,E2 -22251.38} C_VEL
LIN {X 0,Y 195.563,Z 372.348,A -85,B 0,C 180,E1 -22252.683,E2 -22252.683} C_VEL
LIN {X 0,Y 193.718,Z 385.173,A -85,B 0,C 180,E1 -22254.483,E2 -22254.483} C_VEL
LIN {X 0,Y 191.935,Z 395.607,A -85,B 0,C 180,E1 -22256.355,E2 -22256.355} C_VEL
LIN {X 0,Y 190.016,Z 406.171,A -85,B 0,C 180,E1 -22258.736,E2 -22258.736} C_VEL
LIN {X 0,Y 188.095,Z 416.033,A -85,B 0,C 180,E1 -22261.537,E2 -22261.537} C_VEL
LIN {X 0,Y 186.427,Z 424.237,A -85,B 0,C 180,E1 -22264.431,E2 -22264.431} C_VEL
LIN {X 0,Y 185.125,Z 431.016,A -85,B 0,C 180,E1 -22267.398,E2 -22267.398} C_VEL
LIN {X 0,Y 184.037,Z 437.755,A -85,B 0,C 180,E1 -22271.168,E2 -22271.168} C_VEL
LIN {X 0,Y 183.277,Z 442.863,A -85,B 0,C 180,E1 -22274.946,E2 -22274.946} C_VEL
LIN {X 0,Y 182.92,Z 445.942,A -85,B 0,C 180,E1 -22278.026,E2 -22278.026} C_VEL
LIN {X 0,Y 182.969,Z 448.714,A -85,B 0,C 180,E1 -22282.08,E2 -22282.08} C_VEL
LIN {X 0,Y 183.396,Z 449.786,A -85,B 0,C 180,E1 -22284.914,E2 -22284.914} C_VEL
LIN {X 0,Y 184.148,Z 450.235,A -85,B 0,C 180,E1 -22287.704,E2 -22287.704} C_VEL
LIN {X 0,Y 185.3,Z 449.957,A -85,B 0,C 180,E1 -22290.72,E2 -22290.72} C_VEL
LIN {X 0,Y 187.185,Z 448.641,A -85,B 0,C 180,E1 -22294.29,E2 -22294.29} C_VEL
LIN {X 0,Y 190.105,Z 445.719,A -85,B 0,C 180,E1 -22298.304,E2 -22298.304} C_VEL
LIN {X 0,Y 192.893,Z 442.419,A -85,B 0,C 180,E1 -22301.299,E2 -22301.299} C_VEL
LIN {X 0,Y 196.77,Z 437.296,A -85,B 0,C 180,E1 -22304.633,E2 -22304.633} C_VEL
LIN {X 0,Y 201.316,Z 430.553,A -85,B 0,C 180,E1 -22307.91,E2 -22307.91} C_VEL
LIN {X 0,Y 205.74,Z 423.059,A -85,B 0,C 180,E1 -22310.669,E2 -22310.669} C_VEL
LIN {X 0,Y 210.57,Z 414.028,A -85,B 0,C 180,E1 -22313.192,E2 -22313.192} C_VEL
LIN {X 0,Y 215.16,Z 404.231,A -85,B 0,C 180,E1 -22315.317,E2 -22315.317} C_VEL
LIN {X 0,Y 219.318,Z 393.709,A -85,B 0,C 180,E1 -22317.116,E2 -22317.116} C_VEL
LIN {X 0,Y 223.024,Z 382.649,A -85,B 0,C 180,E1 -22318.58,E2 -22318.58} C_VEL
LIN {X 0,Y 226.322,Z 370.453,A -85,B 0,C 180,E1 -22319.816,E2 -22319.816} C_VEL
LIN {X 0,Y 228.771,Z 357.844,A -85,B 0,C 180,E1 -22320.775,E2 -22320.775} C_VEL
LIN {X 0,Y 230.632,Z 344.758,A -85,B 0,C 180,E1 -22321.408,E2 -22321.408} C_VEL
LIN {X 0,Y 234.122,Z 309.777,A -85,B 0,C 180,E1 -22322.688,E2 -22322.688} C_VEL
LIN {X 0,Y 229.209,Z 299.287,A -85,B 0,C 180,E1 -22325.749,E2 -22325.749} C_VEL
LIN {X 0,Y 226.476,Z 294.752,A -85,B 0,C 180,E1 -22327.633,E2 -22327.633} C_VEL
LIN {X 0,Y 223.232,Z 289.819,A -85,B 0,C 180,E1 -22330.173,E2 -22330.173} C_VEL
LIN {X 0,Y 221.066,Z 286.468,A -85,B 0,C 180,E1 -22332.237,E2 -22332.237} C_VEL
LIN {X 0,Y 218.836,Z 283.548,A -85,B 0,C 180,E1 -22334.752,E2 -22334.752} C_VEL
LIN {X 0,Y 216.9,Z 281.198,A -85,B 0,C 180,E1 -22337.609,E2 -22337.609} C_VEL
LIN {X 0,Y 215.466,Z 279.503,A -85,B 0,C 180,E1 -22341.027,E2 -22341.027} C_VEL
LIN {X 0,Y 214.945,Z 279.667,A -85,B 0,C 180,E1 -22345.924,E2 -22345.924} C_VEL
LIN {X 0,Y 215.458,Z 280.851,A -85,B 0,C 180,E1 -22348.807,E2 -22348.807} C_VEL
LIN {X 0,Y 216.445,Z 282.609,A -85,B 0,C 180,E1 -22351.301,E2 -22351.301} C_VEL
LIN {X 0,Y 219.601,Z 288.433,A -85,B 0,C 180,E1 -22356.081,E2 -22356.081} C_VEL
LIN {X 0,Y 222.649,Z 294.268,A -85,B 0,C 180,E1 -22359.227,E2 -22359.227} C_VEL
LIN {X 0,Y 225.473,Z 299.985,A -85,B 0,C 180,E1 -22361.583,E2 -22361.583} C_VEL
LIN {X 0,Y 228.15,Z 305.782,A -85,B 0,C 180,E1 -22363.565,E2 -22363.565} C_VEL
LIN {X 0,Y 231.248,Z 313.55,A -85,B 0,C 180,E1 -22365.659,E2 -22365.659} C_VEL
LIN {X 0,Y 233.09,Z 319.147,A -85,B 0,C 180,E1 -22366.862,E2 -22366.862} C_VEL
LIN {X 0,Y 233.055,Z 324.028,A -85,B 0,C 180,E1 -22367.214,E2 -22367.214} C_VEL
LIN {X 0,Y 231.962,Z 334.832,A -85,B 0,C 180,E1 -22367.596,E2 -22367.596} C_VEL
LIN {X 0,Y 230.993,Z 340.677,A -85,B 0,C 180,E1 -22367.64,E2 -22367.64} C_VEL
LIN {X 0,Y 225.793,Z 359.723,A -85,B 0,C 180,E1 -22367.119,E2 -22367.119} C_VEL
LIN {X 0,Y 224.524,Z 365.452,A -85,B 0,C 180,E1 -22367.265,E2 -22367.265} C_VEL
LIN {X 0,Y 221.647,Z 379.084,A -85,B 0,C 180,E1 -22368.121,E2 -22368.121} C_VEL
LIN {X 0,Y 217.92,Z 391.988,A -85,B 0,C 180,E1 -22369.232,E2 -22369.232} C_VEL
LIN {X 0,Y 213.994,Z 402.859,A -85,B 0,C 180,E1 -22370.488,E2 -22370.488} C_VEL
LIN {X 0,Y 209.252,Z 414.098,A -85,B 0,C 180,E1 -22372.202,E2 -22372.202} C_VEL
LIN {X 0,Y 204.34,Z 424.242,A -85,B 0,C 180,E1 -22374.223,E2 -22374.223} C_VEL
LIN {X 0,Y 198.89,Z 434.094,A -85,B 0,C 180,E1 -22376.794,E2 -22376.794} C_VEL
LIN {X 0,Y 193.924,Z 442.16,A -85,B 0,C 180,E1 -22379.514,E2 -22379.514} C_VEL
